LIN {X 0,Y 359.699,Z 331.885,A -85,B 0,C 180,E1 -13391.93,E2 -13391.93} C_VEL
LIN {X 0,Y 358.635,Z 342.585,A -85,B 0,C 180,E1 -13392.906,E2 -13392.906} C_VEL
LIN {X 0,Y 357.527,Z 352.445,A -85,B 0,C 180,E1 -13394.026,E2 -13394.026} C_VEL
LIN {X 0,Y 356.534,Z 362.461,A -85,B 0,C 180,E1 -13395.444,E2 -13395.444} C_VEL
LIN {X 0,Y 355.478,Z 372.178,A -85,B 0,C 180,E1 -13397.149,E2 -13397.149} C_VEL
LIN {X 0,Y 354.559,Z 379.917,A -85,B 0,C 180,E1 -13398.857,E2 -13398.857} C_VEL
LIN {X 0,Y 354.087,Z 385.232,A -85,B 0,C 180,E1 -13400.287,E2 -13400.287} C_VEL
LIN {X 0,Y 353.658,Z 390.386,A -85,B 0,C 180,E1 -13402.004,E2 -13402.004} C_VEL
LIN {X 0,Y 353.447,Z 394.607,A -85,B 0,C 180,E1 -13403.832,E2 -13403.832} C_VEL
LIN {X 0,Y 353.36,Z 397.364,A -85,B 0,C 180,E1 -13405.437,E2 -13405.437} C_VEL
LIN {X 0,Y 353.319,Z 399.786,A -85,B 0,C 180,E1 -13407.72,E2 -13407.72} C_VEL
LIN {X 0,Y 353.4,Z 400.407,A -85,B 0,C 180,E1 -13408.861,E2 -13408.861} C_VEL
LIN {X 0,Y 353.411,Z 400.626,A -85,B 0,C 180,E1 -13410,E2 -13410} C_VEL
LIN {X 0,Y 353.4,Z 400.405,A -85,B 0,C 180,E1 -13411.14,E2 -13411.14} C_VEL
LIN {X 0,Y 353.283,Z 398.772,A -85,B 0,C 180,E1 -13413.422,E2 -13413.422} C_VEL
LIN {X 0,Y 353.36,Z 397.36,A -85,B 0,C 180,E1 -13414.563,E2 -13414.563} C_VEL
LIN {X 0,Y 353.446,Z 394.601,A -85,B 0,C 180,E1 -13416.167,E2 -13416.167} C_VEL
LIN {X 0,Y 353.654,Z 390.371,A -85,B 0,C 180,E1 -13417.996,E2 -13417.996} C_VEL
LIN {X 0,Y 354.203,Z 384.208,A -85,B 0,C 180,E1 -13419.998,E2 -13419.998} C_VEL
LIN {X 0,Y 354.818,Z 377.479,A -85,B 0,C 180,E1 -13421.714,E2 -13421.714} C_VEL
LIN {X 0,Y 355.819,Z 369.151,A -85,B 0,C 180,E1 -13423.42,E2 -13423.42} C_VEL
LIN {X 0,Y 356.807,Z 360.618,A -85,B 0,C 180,E1 -13424.837,E2 -13424.837} C_VEL
LIN {X 0,Y 357.753,Z 350.071,A -85,B 0,C 180,E1 -13426.257,E2 -13426.257} C_VEL
LIN {X 0,Y 359.082,Z 338.231,A -85,B 0,C 180,E1 -13427.513,E2 -13427.513} C_VEL
LIN {X 0,Y 359.668,Z 330.019,A -85,B 0,C 180,E1 -13428.219,E2 -13428.219} C_VEL
LIN {X 0,Y 358.496,Z 318.284,A -85,B 0,C 180,E1 -13429.127,E2 -13429.127} C_VEL
LIN {X 0,Y 356.685,Z 305.211,A -85,B 0,C 180,E1 -13429.919,E2 -13429.919} C_VEL
LIN {X 0,Y 354.401,Z 292.638,A -85,B 0,C 180,E1 -13430.496,E2 -13430.496} C_VEL
LIN {X 0,Y 354.931,Z 285.811,A -85,B 0,C 180,E1 -13433.871,E2 -13433.871} C_VEL
LIN {X 0,Y 355.677,Z 278.035,A -85,B 0,C 180,E1 -13437.688,E2 -13437.688} C_VEL
LIN {X 0,Y 356.457,Z 270.436,A -85,B 0,C 180,E1 -13441.463,E2 -13441.463} C_VEL
LIN {X 0,Y 357.26,Z 263.905,A -85,B 0,C 180,E1 -13444.785,E2 -13444.785} C_VEL
LIN {X 0,Y 357.475,Z 260.008,A -85,B 0,C 180,E1 -13446.859,E2 -13446.859} C_VEL
LIN {X 0,Y 356.766,Z 254.927,A -85,B 0,C 180,E1 -13449.801,E2 -13449.801} C_VEL
LIN {X 0,Y 355.815,Z 249.673,A -85,B 0,C 180,E1 -13453.045,E2 -13453.045} C_VEL
LIN {X 0,Y 354.798,Z 244.294,A -85,B 0,C 180,E1 -13456.67,E2 -13456.67} C_VEL
LIN {X 0,Y 354.787,Z 244.294,A -85,B 0,C 180,E1 -13460.662,E2 -13460.662} C_VEL
LIN {X 0,Y 354.825,Z 244.287,A -85,B 0,C 180,E1 -13464.301,E2 -13464.301} C_VEL
LIN {X 0,Y 354.79,Z 244.288,A -85,B 0,C 180,E1 -13467.667,E2 -13467.667} C_VEL
LIN {X 0,Y 354.802,Z 244.287,A -85,B 0,C 180,E1 -13471.615,E2 -13471.615} C_VEL
LIN {X 0,Y 354.807,Z 244.286,A -85,B 0,C 180,E1 -13475.42,E2 -13475.42} C_VEL
LIN {X 0,Y 354.83,Z 244.283,A -85,B 0,C 180,E1 -13479.113,E2 -13479.113} C_VEL
LIN {X 0,Y 354.903,Z 244.274,A -85,B 0,C 180,E1 -13482.72,E2 -13482.72} C_VEL
LIN {X 0,Y 354.955,Z 244.27,A -85,B 0,C 180,E1 -13486.255,E2 -13486.255} C_VEL
LIN {X 0,Y 354.955,Z 244.273,A -85,B 0,C 180,E1 -13489.735,E2 -13489.735} C_VEL
LIN {X 0,Y 355.116,Z 244.248,A -85,B 0,C 180,E1 -13493.18,E2 -13493.18} C_VEL
LIN {X 0,Y 355.248,Z 244.235,A -85,B 0,C 180,E1 -13497.732,E2 -13497.732} C_VEL
LIN {X 0,Y 355.235,Z 244.232,A -85,B 0,C 180,E1 -13502.268,E2 -13502.268} C_VEL
LIN {X 0,Y 355.116,Z 244.249,A -85,B 0,C 180,E1 -13506.82,E2 -13506.82} C_VEL
LIN {X 0,Y 354.961,Z 244.266,A -85,B 0,C 180,E1 -13510.265,E2 -13510.265} C_VEL
LIN {X 0,Y 354.947,Z 244.268,A -85,B 0,C 180,E1 -13514.019,E2 -13514.019} C_VEL
LIN {X 0,Y 354.894,Z 244.275,A -85,B 0,C 180,E1 -13518.092,E2 -13518.092} C_VEL
LIN {X 0,Y 354.819,Z 244.285,A -85,B 0,C 180,E1 -13522.107,E2 -13522.107} C_VEL
LIN {X 0,Y 354.824,Z 244.283,A -85,B 0,C 180,E1 -13525.833,E2 -13525.833} C_VEL
LIN {X 0,Y 354.799,Z 244.287,A -85,B 0,C 180,E1 -13529.684,E2 -13529.684} C_VEL
LIN {X 0,Y 354.79,Z 244.292,A -85,B 0,C 180,E1 -13532.333,E2 -13532.333} C_VEL
LIN {X 0,Y 354.825,Z 244.284,A -85,B 0,C 180,E1 -13535.699,E2 -13535.699} C_VEL
LIN {X 0,Y 354.827,Z 244.283,A -85,B 0,C 180,E1 -13539.423,E2 -13539.423} C_VEL
LIN {X 0,Y 354.791,Z 244.288,A -85,B 0,C 180,E1 -13542.867,E2 -13542.867} C_VEL
LIN {X 0,Y 354.77,Z 244.296,A -85,B 0,C 180,E1 -13546.104,E2 -13546.104} C_VEL
LIN {X 0,Y 354.787,Z 244.288,A -85,B 0,C 180,E1 -13549.178,E2 -13549.178} C_VEL
LIN {X 0,Y 354.792,Z 244.289,A -85,B 0,C 180,E1 -13552.406,E2 -13552.406} C_VEL
LIN {X 0,Y 354.645,Z 244.306,A -85,B 0,C 180,E1 -13554.921,E2 -13554.921} C_VEL
LIN {X 0,Y 354.359,Z 244.347,A -85,B 0,C 180,E1 -13557.622,E2 -13557.622} C_VEL
LIN {X 0,Y 354.278,Z 245.084,A -85,B 0,C 180,E1 -13558.95,E2 -13558.95} C_VEL
LIN {X 0,Y 354.196,Z 247.346,A -85,B 0,C 180,E1 -13561.561,E2 -13561.561} C_VEL
LIN {X 0,Y 354.111,Z 249.638,A -85,B 0,C 180,E1 -13564.111,E2 -13564.111} C_VEL
LIN {X 0,Y 354.05,Z 251.97,A -85,B 0,C 180,E1 -13566.609,E2 -13566.609} C_VEL
LIN {X 0,Y 354.016,Z 254.952,A -85,B 0,C 180,E1 -13569.596,E2 -13569.596} C_VEL
LIN {X 0,Y 357.921,Z 268.382,A -85,B 0,C 180,E1 -13570.374,E2 -13570.374} C_VEL
LIN {X 0,Y 360.714,Z 280.036,A -85,B 0,C 180,E1 -13571.221,E2 -13571.221} C_VEL
LIN {X 0,Y 361.289,Z 284.038,A -85,B 0,C 180,E1 -13571.541,E2 -13571.541} C_VEL
LIN {X 0,Y 360.357,Z 296.417,A -85,B 0,C 180,E1 -13572.551,E2 -13572.551} C_VEL
LIN {X 0,Y 359.482,Z 306.713,A -85,B 0,C 180,E1 -13573.635,E2 -13573.635} C_VEL
LIN {X 0,Y 358.447,Z 316.732,A -85,B 0,C 180,E1 -13574.942,E2 -13574.942} C_VEL
LIN {X 0,Y 357.377,Z 325.539,A -85,B 0,C 180,E1 -13576.35,E2 -13576.35} C_VEL
LIN {X 0,Y 356.259,Z 334.126,A -85,B 0,C 180,E1 -13578.045,E2 -13578.045} C_VEL
LIN {X 0,Y 355.393,Z 340.963,A -85,B 0,C 180,E1 -13579.748,E2 -13579.748} C_VEL
LIN {X 0,Y 354.749,Z 346.43,A -85,B 0,C 180,E1 -13581.455,E2 -13581.455} C_VEL
LIN {X 0,Y 354.307,Z 350.717,A -85,B 0,C 180,E1 -13583.164,E2 -13583.164} C_VEL
LIN {X 0,Y 353.962,Z 352.992,A -85,B 0,C 180,E1 -13584.302,E2 -13584.302} C_VEL
LIN {X 0,Y 353.832,Z 354.833,A -85,B 0,C 180,E1 -13585.443,E2 -13585.443} C_VEL
LIN {X 0,Y 353.805,Z 356.215,A -85,B 0,C 180,E1 -13586.583,E2 -13586.583} C_VEL
LIN {X 0,Y 353.512,Z 357.818,A -85,B 0,C 180,E1 -13588.861,E2 -13588.861} C_VEL
LIN {X 0,Y 353.483,Z 358.049,A -85,B 0,C 180,E1 -13590,E2 -13590} C_VEL
LIN {X 0,Y 353.634,Z 357.275,A -85,B 0,C 180,E1 -13592.278,E2 -13592.278} C_VEL
LIN {X 0,Y 353.783,Z 356.312,A -85,B 0,C 180,E1 -13593.416,E2 -13593.416} C_VEL
LIN {X 0,Y 353.822,Z 354.972,A -85,B 0,C 180,E1 -13594.557,E2 -13594.557} C_VEL
LIN {X 0,Y 354.111,Z 352.127,A -85,B 0,C 180,E1 -13596.267,E2 -13596.267} C_VEL
LIN {X 0,Y 354.551,Z 348.265,A -85,B 0,C 180,E1 -13597.976,E2 -13597.976} C_VEL
LIN {X 0,Y 355.108,Z 343.282,A -85,B 0,C 180,E1 -13599.685,E2 -13599.685} C_VEL
LIN {X 0,Y 355.96,Z 336.996,A -85,B 0,C 180,E1 -13601.387,E2 -13601.387} C_VEL
LIN {X 0,Y 356.932,Z 329.129,A -85,B 0,C 180,E1 -13603.087,E2 -13603.087} C_VEL
LIN {X 0,Y 357.867,Z 321.104,A -85,B 0,C 180,E1 -13604.501,E2 -13604.501} C_VEL
LIN {X 0,Y 358.993,Z 311.302,A -85,B 0,C 180,E1 -13605.907,E2 -13605.907} C_VEL
LIN {X 0,Y 359.9,Z 301.655,A -85,B 0,C 180,E1 -13607.032,E2 -13607.032} C_VEL
LIN {X 0,Y 360.833,Z 291.2,A -85,B 0,C 180,E1 -13608.011,E2 -13608.011} C_VEL
LIN {X 0,Y 361.263,Z 282.387,A -85,B 0,C 180,E1 -13608.688,E2 -13608.688} C_VEL
LIN {X 0,Y 358.303,Z 269.681,A -85,B 0,C 180,E1 -13609.644,E2 -13609.644} C_VEL
LIN {X 0,Y 354.312,Z 256.261,A -85,B 0,C 180,E1 -13610.444,E2 -13610.444} C_VEL
LIN {X 0,Y 354.04,Z 254.897,A -85,B 0,C 180,E1 -13610.509,E2 -13610.509} C_VEL
LIN {X 0,Y 354.071,Z 250.911,A -85,B 0,C 180,E1 -13614.635,E2 -13614.635} C_VEL
LIN {X 0,Y 354.183,Z 247.453,A -85,B 0,C 180,E1 -13618.439,E2 -13618.439} C_VEL
LIN {X 0,Y 354.294,Z 244.842,A -85,B 0,C 180,E1 -13621.463,E2 -13621.463} C_VEL
LIN {X 0,Y 354.342,Z 244.351,A -85,B 0,C 180,E1 -13622.379,E2 -13622.379} C_VEL
LIN {X 0,Y 354.712,Z 244.299,A -85,B 0,C 180,E1 -13625.674,E2 -13625.674} C_VEL
LIN {X 0,Y 354.763,Z 244.292,A -85,B 0,C 180,E1 -13627.302,E2 -13627.302} C_VEL
LIN {X 0,Y 354.156,Z 244.373,A -85,B 0,C 180,E1 -13628.25,E2 -13628.25} C_VEL
LIN {X 0,Y 351.326,Z 244.724,A -85,B 0,C 180,E1 -13629.791,E2 -13629.791} C_VEL
LIN {X 0,Y 348.881,Z 245.028,A -85,B 0,C 180,E1 -13631.038,E2 -13631.038} C_VEL
LIN {X 0,Y 347.812,Z 245.162,A -85,B 0,C 180,E1 -13632.003,E2 -13632.003} C_VEL
LIN {X 0,Y 347.717,Z 245.168,A -85,B 0,C 180,E1 -13632.33,E2 -13632.33} C_VEL
LIN {X 0,Y 347.707,Z 245.17,A -85,B 0,C 180,E1 -13635.027,E2 -13635.027} C_VEL
LIN {X 0,Y 347.751,Z 245.166,A -85,B 0,C 180,E1 -13638.397,E2 -13638.397} C_VEL
LIN {X 0,Y 347.774,Z 245.165,A -85,B 0,C 180,E1 -13642.011,E2 -13642.011} C_VEL
LIN {X 0,Y 347.746,Z 245.17,A -85,B 0,C 180,E1 -13645.536,E2 -13645.536} C_VEL
LIN {X 0,Y 347.748,Z 245.165,A -85,B 0,C 180,E1 -13648.301,E2 -13648.301} C_VEL
LIN {X 0,Y 347.747,Z 245.166,A -85,B 0,C 180,E1 -13650.985,E2 -13650.985} C_VEL
LIN {X 0,Y 347.752,Z 245.168,A -85,B 0,C 180,E1 -13653.601,E2 -13653.601} C_VEL
LIN {X 0,Y 347.772,Z 245.162,A -85,B 0,C 180,E1 -13656.161,E2 -13656.161} C_VEL
LIN {X 0,Y 347.802,Z 245.159,A -85,B 0,C 180,E1 -13659.909,E2 -13659.909} C_VEL
LIN {X 0,Y 347.833,Z 245.156,A -85,B 0,C 180,E1 -13663.568,E2 -13663.568} C_VEL
LIN {X 0,Y 347.893,Z 245.151,A -85,B 0,C 180,E1 -13667.161,E2 -13667.161} C_VEL
LIN {X 0,Y 348.096,Z 245.122,A -85,B 0,C 180,E1 -13671.612,E2 -13671.612} C_VEL
LIN {X 0,Y 348.067,Z 245.126,A -85,B 0,C 180,E1 -13674.206,E2 -13674.206} C_VEL
LIN {X 0,Y 348.196,Z 245.109,A -85,B 0,C 180,E1 -13677.686,E2 -13677.686} C_VEL
LIN {X 0,Y 348.147,Z 245.116,A -85,B 0,C 180,E1 -13681.157,E2 -13681.157} C_VEL
LIN {X 0,Y 348.208,Z 245.112,A -85,B 0,C 180,E1 -13682.313,E2 -13682.313} C_VEL
LIN {X 0,Y 348.08,Z 245.124,A -85,B 0,C 180,E1 -13686.958,E2 -13686.958} C_VEL
LIN {X 0,Y 347.895,Z 245.15,A -85,B 0,C 180,E1 -13690.475,E2 -13690.475} C_VEL
LIN {X 0,Y 347.901,Z 245.152,A -85,B 0,C 180,E1 -13694.15,E2 -13694.15} C_VEL
LIN {X 0,Y 347.894,Z 245.15,A -85,B 0,C 180,E1 -13698.291,E2 -13698.291} C_VEL
LIN {X 0,Y 347.766,Z 245.166,A -85,B 0,C 180,E1 -13701.625,E2 -13701.625} C_VEL
LIN {X 0,Y 347.739,Z 245.167,A -85,B 0,C 180,E1 -13705.114,E2 -13705.114} C_VEL
LIN {X 0,Y 347.737,Z 245.173,A -85,B 0,C 180,E1 -13707.7,E2 -13707.7} C_VEL
LIN {X 0,Y 347.742,Z 245.167,A -85,B 0,C 180,E1 -13710.349,E2 -13710.349} C_VEL
LIN {X 0,Y 347.75,Z 245.167,A -85,B 0,C 180,E1 -13714.044,E2 -13714.044} C_VEL
LIN {X 0,Y 347.757,Z 245.17,A -85,B 0,C 180,E1 -13717.321,E2 -13717.321} C_VEL
LIN {X 0,Y 347.742,Z 245.169,A -85,B 0,C 180,E1 -13721.601,E2 -13721.601} C_VEL
LIN {X 0,Y 347.769,Z 245.276,A -85,B 0,C 180,E1 -13722.971,E2 -13722.971} C_VEL
LIN {X 0,Y 348.742,Z 250.485,A -85,B 0,C 180,E1 -13726.51,E2 -13726.51} C_VEL
LIN {X 0,Y 349.745,Z 256,A -85,B 0,C 180,E1 -13729.982,E2 -13729.982} C_VEL
LIN {X 0,Y 350.464,Z 261.145,A -85,B 0,C 180,E1 -13733.015,E2 -13733.015} C_VEL
LIN {X 0,Y 350.204,Z 265.441,A -85,B 0,C 180,E1 -13735.366,E2 -13735.366} C_VEL
LIN {X 0,Y 349.297,Z 272.644,A -85,B 0,C 180,E1 -13739.131,E2 -13739.131} C_VEL
LIN {X 0,Y 348.563,Z 279.286,A -85,B 0,C 180,E1 -13742.519,E2 -13742.519} C_VEL
LIN {X 0,Y 347.839,Z 286.516,A -85,B 0,C 180,E1 -13746.166,E2 -13746.166} C_VEL
LIN {X 0,Y 347.376,Z 292.278,A -85,B 0,C 180,E1 -13749.071,E2 -13749.071} C_VEL
LIN {X 0,Y 349.887,Z 305.889,A -85,B 0,C 180,E1 -13749.717,E2 -13749.717} C_VEL
LIN {X 0,Y 351.591,Z 318.635,A -85,B 0,C 180,E1 -13750.527,E2 -13750.527} C_VEL
LIN {X 0,Y 352.663,Z 329.662,A -85,B 0,C 180,E1 -13751.406,E2 -13751.406} C_VEL
LIN {X 0,Y 352.791,Z 333.152,A -85,B 0,C 180,E1 -13751.714,E2 -13751.714} C_VEL
LIN {X 0,Y 351.522,Z 344.774,A -85,B 0,C 180,E1 -13752.849,E2 -13752.849} C_VEL
LIN {X 0,Y 350.29,Z 355.459,A -85,B 0,C 180,E1 -13754.165,E2 -13754.165} C_VEL
LIN {X 0,Y 349.416,Z 363.829,A -85,B 0,C 180,E1 -13755.439,E2 -13755.439} C_VEL
LIN {X 0,Y 348.53,Z 371.751,A -85,B 0,C 180,E1 -13756.888,E2 -13756.888} C_VEL
LIN {X 0,Y 347.551,Z 379.488,A -85,B 0,C 180,E1 -13758.629,E2 -13758.629} C_VEL
LIN {X 0,Y 347.071,Z 384.804,A -85,B 0,C 180,E1 -13760.089,E2 -13760.089} C_VEL
LIN {X 0,Y 346.594,Z 389.958,A -85,B 0,C 180,E1 -13761.84,E2 -13761.84} C_VEL
LIN {X 0,Y 346.343,Z 394.513,A -85,B 0,C 180,E1 -13763.886,E2 -13763.886} C_VEL
LIN {X 0,Y 346.274,Z 396.936,A -85,B 0,C 180,E1 -13765.344,E2 -13765.344} C_VEL
LIN {X 0,Y 346.224,Z 399.358,A -85,B 0,C 180,E1 -13767.673,E2 -13767.673} C_VEL
LIN {X 0,Y 346.32,Z 399.98,A -85,B 0,C 180,E1 -13768.837,E2 -13768.837} C_VEL
LIN {X 0,Y 346.35,Z 400.2,A -85,B 0,C 180,E1 -13770,E2 -13770} C_VEL
LIN {X 0,Y 346.32,Z 399.978,A -85,B 0,C 180,E1 -13771.163,E2 -13771.163} C_VEL
LIN {X 0,Y 346.206,Z 398.345,A -85,B 0,C 180,E1 -13773.492,E2 -13773.492} C_VEL
LIN {X 0,Y 346.274,Z 396.932,A -85,B 0,C 180,E1 -13774.657,E2 -13774.657} C_VEL
LIN {X 0,Y 346.343,Z 394.506,A -85,B 0,C 180,E1 -13776.113,E2 -13776.113} C_VEL
LIN {X 0,Y 346.592,Z 389.94,A -85,B 0,C 180,E1 -13778.16,E2 -13778.16} C_VEL
LIN {X 0,Y 347.172,Z 383.777,A -85,B 0,C 180,E1 -13780.203,E2 -13780.203} C_VEL
LIN {X 0,Y 347.831,Z 377.048,A -85,B 0,C 180,E1 -13781.953,E2 -13781.953} C_VEL
LIN {X 0,Y 348.846,Z 368.717,A -85,B 0,C 180,E1 -13783.693,E2 -13783.693} C_VEL
LIN {X 0,Y 350.015,Z 359.161,A -85,B 0,C 180,E1 -13785.288,E2 -13785.288} C_VEL
LIN {X 0,Y 350.909,Z 349.638,A -85,B 0,C 180,E1 -13786.583,E2 -13786.583} C_VEL
LIN {X 0,Y 352.317,Z 337.799,A -85,B 0,C 180,E1 -13787.861,E2 -13787.861} C_VEL
LIN {X 0,Y 352.813,Z 331.363,A -85,B 0,C 180,E1 -13788.435,E2 -13788.435} C_VEL
LIN {X 0,Y 351.787,Z 320.21,A -85,B 0,C 180,E1 -13789.349,E2 -13789.349} C_VEL
LIN {X 0,Y 350.003,Z 306.683,A -85,B 0,C 180,E1 -13790.228,E2 -13790.228} C_VEL
LIN {X 0,Y 347.564,Z 293.686,A -85,B 0,C 180,E1 -13790.869,E2 -13790.869} C_VEL
LIN {X 0,Y 347.392,Z 292.22,A -85,B 0,C 180,E1 -13790.919,E2 -13790.919} C_VEL
LIN {X 0,Y 348.091,Z 283.999,A -85,B 0,C 180,E1 -13795.087,E2 -13795.087} C_VEL
LIN {X 0,Y 348.873,Z 276.433,A -85,B 0,C 180,E1 -13798.913,E2 -13798.913} C_VEL
LIN {X 0,Y 349.772,Z 268.732,A -85,B 0,C 180,E1 -13802.855,E2 -13802.855} C_VEL
LIN {X 0,Y 350.378,Z 263.584,A -85,B 0,C 180,E1 -13805.57,E2 -13805.57} C_VEL
LIN {X 0,Y 350.337,Z 259.724,A -85,B 0,C 180,E1 -13807.724,E2 -13807.724} C_VEL
LIN {X 0,Y 349.539,Z 254.573,A -85,B 0,C 180,E1 -13810.835,E2 -13810.835} C_VEL
LIN {X 0,Y 348.371,Z 248.298,A -85,B 0,C 180,E1 -13814.918,E2 -13814.918} C_VEL
LIN {X 0,Y 347.755,Z 245.17,A -85,B 0,C 180,E1 -13817.219,E2 -13817.219} C_VEL
LIN {X 0,Y 347.733,Z 245.168,A -85,B 0,C 180,E1 -13821.205,E2 -13821.205} C_VEL
LIN {X 0,Y 347.791,Z 245.162,A -85,B 0,C 180,E1 -13824.125,E2 -13824.125} C_VEL
LIN {X 0,Y 347.742,Z 245.169,A -85,B 0,C 180,E1 -13828.086,E2 -13828.086} C_VEL
LIN {X 0,Y 347.748,Z 245.166,A -85,B 0,C 180,E1 -13830.985,E2 -13830.985} C_VEL
LIN {X 0,Y 347.745,Z 245.166,A -85,B 0,C 180,E1 -13833.601,E2 -13833.601} C_VEL
LIN {X 0,Y 347.752,Z 245.171,A -85,B 0,C 180,E1 -13836.159,E2 -13836.159} C_VEL
LIN {X 0,Y 347.812,Z 245.162,A -85,B 0,C 180,E1 -13839.909,E2 -13839.909} C_VEL
LIN {X 0,Y 347.87,Z 245.153,A -85,B 0,C 180,E1 -13842.359,E2 -13842.359} C_VEL
LIN {X 0,Y 347.901,Z 245.151,A -85,B 0,C 180,E1 -13845.971,E2 -13845.971} C_VEL
LIN {X 0,Y 347.895,Z 245.15,A -85,B 0,C 180,E1 -13849.525,E2 -13849.525} C_VEL
LIN {X 0,Y 348.082,Z 245.124,A -85,B 0,C 180,E1 -13853.042,E2 -13853.042} C_VEL
LIN {X 0,Y 348.21,Z 245.112,A -85,B 0,C 180,E1 -13857.687,E2 -13857.687} C_VEL
LIN {X 0,Y 348.121,Z 245.121,A -85,B 0,C 180,E1 -13861.157,E2 -13861.157} C_VEL
LIN {X 0,Y 348.197,Z 245.109,A -85,B 0,C 180,E1 -13862.314,E2 -13862.314} C_VEL
LIN {X 0,Y 348.082,Z 245.126,A -85,B 0,C 180,E1 -13866.958,E2 -13866.958} C_VEL
LIN {X 0,Y 347.901,Z 245.146,A -85,B 0,C 180,E1 -13870.475,E2 -13870.475} C_VEL
LIN {X 0,Y 347.903,Z 245.146,A -85,B 0,C 180,E1 -13874.15,E2 -13874.15} C_VEL
LIN {X 0,Y 347.833,Z 245.155,A -85,B 0,C 180,E1 -13878.259,E2 -13878.259} C_VEL
LIN {X 0,Y 347.771,Z 245.162,A -85,B 0,C 180,E1 -13881.626,E2 -13881.626} C_VEL
LIN {X 0,Y 347.776,Z 245.163,A -85,B 0,C 180,E1 -13885.111,E2 -13885.111} C_VEL
LIN {X 0,Y 347.741,Z 245.166,A -85,B 0,C 180,E1 -13887.7,E2 -13887.7} C_VEL
LIN {X 0,Y 347.741,Z 245.17,A -85,B 0,C 180,E1 -13890.349,E2 -13890.349} C_VEL
LIN {X 0,Y 347.752,Z 245.167,A -85,B 0,C 180,E1 -13894.044,E2 -13894.044} C_VEL
LIN {X 0,Y 347.764,Z 245.163,A -85,B 0,C 180,E1 -13897.321,E2 -13897.321} C_VEL
LIN {X 0,Y 347.735,Z 245.172,A -85,B 0,C 180,E1 -13900.297,E2 -13900.297} C_VEL
LIN {X 0,Y 347.726,Z 245.168,A -85,B 0,C 180,E1 -13903.408,E2 -13903.408} C_VEL
LIN {X 0,Y 347.728,Z 245.168,A -85,B 0,C 180,E1 -13906.686,E2 -13906.686} C_VEL
LIN {X 0,Y 347.749,Z 245.168,A -85,B 0,C 180,E1 -13910.173,E2 -13910.173} C_VEL
LIN {X 0,Y 347.739,Z 245.166,A -85,B 0,C 180,E1 -13912.676,E2 -13912.676} C_VEL
LIN {X 0,Y 347.486,Z 245.202,A -85,B 0,C 180,E1 -13916.021,E2 -13916.021} C_VEL
LIN {X 0,Y 347.269,Z 245.446,A -85,B 0,C 180,E1 -13918.252,E2 -13918.252} C_VEL
LIN {X 0,Y 347.192,Z 247.715,A -85,B 0,C 180,E1 -13920.934,E2 -13920.934} C_VEL
LIN {X 0,Y 347.103,Z 250.029,A -85,B 0,C 180,E1 -13923.548,E2 -13923.548} C_VEL
LIN {X 0,Y 347.045,Z 252.379,A -85,B 0,C 180,E1 -13926.107,E2 -13926.107} C_VEL
LIN {X 0,Y 347.001,Z 255.445,A -85,B 0,C 180,E1 -13929.169,E2 -13929.169} C_VEL
LIN {X 0,Y 350.855,Z 268.565,A -85,B 0,C 180,E1 -13929.948,E2 -13929.948} C_VEL
LIN {X 0,Y 353.896,Z 280.989,A -85,B 0,C 180,E1 -13930.879,E2 -13930.879} C_VEL
LIN {X 0,Y 354.572,Z 284.714,A -85,B 0,C 180,E1 -13931.197,E2 -13931.197} C_VEL
LIN {X 0,Y 353.624,Z 296.848,A -85,B 0,C 180,E1 -13932.207,E2 -13932.207} C_VEL
LIN {X 0,Y 352.659,Z 307.491,A -85,B 0,C 180,E1 -13933.354,E2 -13933.354} C_VEL
LIN {X 0,Y 351.608,Z 317.162,A -85,B 0,C 180,E1 -13934.642,E2 -13934.642} C_VEL
LIN {X 0,Y 350.477,Z 325.969,A -85,B 0,C 180,E1 -13936.076,E2 -13936.076} C_VEL
LIN {X 0,Y 349.336,Z 334.554,A -85,B 0,C 180,E1 -13937.805,E2 -13937.805} C_VEL
LIN {X 0,Y 348.421,Z 341.391,A -85,B 0,C 180,E1 -13939.54,E2 -13939.54} C_VEL
LIN {X 0,Y 347.756,Z 346.858,A -85,B 0,C 180,E1 -13941.282,E2 -13941.282} C_VEL
LIN {X 0,Y 347.282,Z 351.145,A -85,B 0,C 180,E1 -13943.026,E2 -13943.026} C_VEL
LIN {X 0,Y 346.926,Z 353.419,A -85,B 0,C 180,E1 -13944.186,E2 -13944.186} C_VEL
LIN {X 0,Y 346.759,Z 355.261,A -85,B 0,C 180,E1 -13945.35,E2 -13945.35} C_VEL
LIN {X 0,Y 346.735,Z 356.642,A -85,B 0,C 180,E1 -13946.514,E2 -13946.514} C_VEL
LIN {X 0,Y 346.45,Z 358.243,A -85,B 0,C 180,E1 -13948.837,E2 -13948.837} C_VEL
LIN {X 0,Y 346.419,Z 358.475,A -85,B 0,C 180,E1 -13950,E2 -13950} C_VEL
LIN {X 0,Y 346.579,Z 357.7,A -85,B 0,C 180,E1 -13952.324,E2 -13952.324} C_VEL
LIN {X 0,Y 346.714,Z 356.738,A -85,B 0,C 180,E1 -13953.486,E2 -13953.486} C_VEL
LIN {X 0,Y 346.748,Z 355.399,A -85,B 0,C 180,E1 -13954.65,E2 -13954.65} C_VEL
LIN {X 0,Y 347.083,Z 352.551,A -85,B 0,C 180,E1 -13956.394,E2 -13956.394} C_VEL
LIN {X 0,Y 347.524,Z 348.691,A -85,B 0,C 180,E1 -13958.138,E2 -13958.138} C_VEL
LIN {X 0,Y 348.111,Z 343.708,A -85,B 0,C 180,E1 -13959.881,E2 -13959.881} C_VEL
LIN {X 0,Y 349.017,Z 337.421,A -85,B 0,C 180,E1 -13961.617,E2 -13961.617} C_VEL
LIN {X 0,Y 350.044,Z 329.552,A -85,B 0,C 180,E1 -13963.349,E2 -13963.349} C_VEL
LIN {X 0,Y 351.019,Z 321.527,A -85,B 0,C 180,E1 -13964.79,E2 -13964.79} C_VEL
LIN {X 0,Y 352.19,Z 311.724,A -85,B 0,C 180,E1 -13966.223,E2 -13966.223} C_VEL
LIN {X 0,Y 353.129,Z 302.077,A -85,B 0,C 180,E1 -13967.369,E2 -13967.369} C_VEL
LIN {X 0,Y 354.113,Z 291.619,A -85,B 0,C 180,E1 -13968.365,E2 -13968.365} C_VEL
LIN {X 0,Y 354.608,Z 284.317,A -85,B 0,C 180,E1 -13968.936,E2 -13968.936} C_VEL
LIN {X 0,Y 351.729,Z 271.686,A -85,B 0,C 180,E1 -13969.944,E2 -13969.944} C_VEL
LIN {X 0,Y 348.006,Z 258.847,A -85,B 0,C 180,E1 -13970.757,E2 -13970.757} C_VEL
LIN {X 0,Y 346.974,Z 255.305,A -85,B 0,C 180,E1 -13970.967,E2 -13970.967} C_VEL
LIN {X 0,Y 347.039,Z 252.095,A -85,B 0,C 180,E1 -13974.312,E2 -13974.312} C_VEL
LIN {X 0,Y 347.104,Z 248.978,A -85,B 0,C 180,E1 -13977.755,E2 -13977.755} C_VEL
LIN {X 0,Y 347.197,Z 246.68,A -85,B 0,C 180,E1 -13980.401,E2 -13980.401} C_VEL
LIN {X 0,Y 347.252,Z 245.516,A -85,B 0,C 180,E1 -13981.784,E2 -13981.784} C_VEL
LIN {X 0,Y 347.549,Z 245.195,A -85,B 0,C 180,E1 -13984.486,E2 -13984.486} C_VEL
LIN {X 0,Y 347.738,Z 245.167,A -85,B 0,C 180,E1 -13987.324,E2 -13987.324} C_VEL
LIN {X 0,Y 347.734,Z 245.171,A -85,B 0,C 180,E1 -13990.297,E2 -13990.297} C_VEL
LIN {X 0,Y 347.717,Z 245.168,A -85,B 0,C 180,E1 -13992.33,E2 -13992.33} C_VEL
LIN {X 0,Y 347.027,Z 245.256,A -85,B 0,C 180,E1 -13993.297,E2 -13993.297} C_VEL
LIN {X 0,Y 344.165,Z 245.612,A -85,B 0,C 180,E1 -13994.87,E2 -13994.87} C_VEL
LIN {X 0,Y 341.766,Z 245.914,A -85,B 0,C 180,E1 -13996.143,E2 -13996.143} C_VEL
LIN {X 0,Y 340.752,Z 246.036,A -85,B 0,C 180,E1 -13997.128,E2 -13997.128} C_VEL
LIN {X 0,Y 340.678,Z 246.047,A -85,B 0,C 180,E1 -13997.462,E2 -13997.462} C_VEL
LIN {X 0,Y 340.701,Z 246.045,A -85,B 0,C 180,E1 -14000.247,E2 -14000.247} C_VEL
LIN {X 0,Y 340.712,Z 246.046,A -85,B 0,C 180,E1 -14003.559,E2 -14003.559} C_VEL
LIN {X 0,Y 340.696,Z 246.045,A -85,B 0,C 180,E1 -14006.154,E2 -14006.154} C_VEL
LIN {X 0,Y 340.725,Z 246.041,A -85,B 0,C 180,E1 -14010.034,E2 -14010.034} C_VEL
LIN {X 0,Y 340.722,Z 246.042,A -85,B 0,C 180,E1 -14013.013,E2 -14013.013} C_VEL
LIN {X 0,Y 340.743,Z 246.041,A -85,B 0,C 180,E1 -14015.637,E2 -14015.637} C_VEL
LIN {X 0,Y 340.732,Z 246.042,A -85,B 0,C 180,E1 -14019.473,E2 -14019.473} C_VEL
LIN {X 0,Y 340.794,Z 246.031,A -85,B 0,C 180,E1 -14021.981,E2 -14021.981} C_VEL
LIN {X 0,Y 340.871,Z 246.022,A -85,B 0,C 180,E1 -14025.705,E2 -14025.705} C_VEL
LIN {X 0,Y 340.874,Z 246.023,A -85,B 0,C 180,E1 -14029.306,E2 -14029.306} C_VEL
LIN {X 0,Y 341.077,Z 246.001,A -85,B 0,C 180,E1 -14032.898,E2 -14032.898} C_VEL
LIN {X 0,Y 341.133,Z 245.989,A -85,B 0,C 180,E1 -14037.638,E2 -14037.638} C_VEL
LIN {X 0,Y 341.116,Z 245.992,A -85,B 0,C 180,E1 -14041.18,E2 -14041.18} C_VEL
LIN {X 0,Y 341.17,Z 245.989,A -85,B 0,C 180,E1 -14042.361,E2 -14042.361} C_VEL
LIN {X 0,Y 341.048,Z 246,A -85,B 0,C 180,E1 -14047.102,E2 -14047.102} C_VEL
LIN {X 0,Y 340.847,Z 246.027,A -85,B 0,C 180,E1 -14050.695,E2 -14050.695} C_VEL
LIN {X 0,Y 340.865,Z 246.026,A -85,B 0,C 180,E1 -14054.325,E2 -14054.325} C_VEL
LIN {X 0,Y 340.84,Z 246.027,A -85,B 0,C 180,E1 -14058.467,E2 -14058.467} C_VEL
LIN {X 0,Y 340.719,Z 246.046,A -85,B 0,C 180,E1 -14061.842,E2 -14061.842} C_VEL
LIN {X 0,Y 340.676,Z 246.052,A -85,B 0,C 180,E1 -14065.672,E2 -14065.672} C_VEL
LIN {X 0,Y 340.683,Z 246.047,A -85,B 0,C 180,E1 -14068.325,E2 -14068.325} C_VEL
LIN {X 0,Y 340.696,Z 246.046,A -85,B 0,C 180,E1 -14071.045,E2 -14071.045} C_VEL
LIN {X 0,Y 340.719,Z 246.046,A -85,B 0,C 180,E1 -14075.279,E2 -14075.279} C_VEL
LIN {X 0,Y 340.695,Z 246.045,A -85,B 0,C 180,E1 -14078.382,E2 -14078.382} C_VEL
LIN {X 0,Y 340.731,Z 246.075,A -85,B 0,C 180,E1 -14082.418,E2 -14082.418} C_VEL
LIN {X 0,Y 341.688,Z 251.245,A -85,B 0,C 180,E1 -14086.046,E2 -14086.046} C_VEL
LIN {X 0,Y 342.631,Z 256.348,A -85,B 0,C 180,E1 -14089.371,E2 -14089.371} C_VEL
LIN {X 0,Y 343.328,Z 260.832,A -85,B 0,C 180,E1 -14092.113,E2 -14092.113} C_VEL
LIN {X 0,Y 343.385,Z 264.665,A -85,B 0,C 180,E1 -14094.317,E2 -14094.317} C_VEL
LIN {X 0,Y 342.556,Z 271.031,A -85,B 0,C 180,E1 -14097.763,E2 -14097.763} C_VEL
LIN {X 0,Y 341.678,Z 278.627,A -85,B 0,C 180,E1 -14101.765,E2 -14101.765} C_VEL
LIN {X 0,Y 340.864,Z 286.115,A -85,B 0,C 180,E1 -14105.647,E2 -14105.647} C_VEL
LIN {X 0,Y 340.39,Z 291.854,A -85,B 0,C 180,E1 -14108.62,E2 -14108.62} C_VEL
LIN {X 0,Y 342.92,Z 305.591,A -85,B 0,C 180,E1 -14109.294,E2 -14109.294} C_VEL
LIN {X 0,Y 344.647,Z 318.238,A -85,B 0,C 180,E1 -14110.121,E2 -14110.121} C_VEL
LIN {X 0,Y 345.847,Z 331.016,A -85,B 0,C 180,E1 -14111.18,E2 -14111.18} C_VEL
LIN {X 0,Y 345.707,Z 335.904,A -85,B 0,C 180,E1 -14111.633,E2 -14111.633} C_VEL
LIN {X 0,Y 344.426,Z 346.912,A -85,B 0,C 180,E1 -14112.79,E2 -14112.79} C_VEL
LIN {X 0,Y 343.268,Z 356.263,A -85,B 0,C 180,E1 -14114.016,E2 -14114.016} C_VEL
LIN {X 0,Y 342.291,Z 365.088,A -85,B 0,C 180,E1 -14115.433,E2 -14115.433} C_VEL
LIN {X 0,Y 341.208,Z 374.076,A -85,B 0,C 180,E1 -14117.207,E2 -14117.207} C_VEL
LIN {X 0,Y 340.345,Z 381.316,A -85,B 0,C 180,E1 -14118.988,E2 -14118.988} C_VEL
LIN {X 0,Y 339.846,Z 386.212,A -85,B 0,C 180,E1 -14120.477,E2 -14120.477} C_VEL
LIN {X 0,Y 339.445,Z 390.977,A -85,B 0,C 180,E1 -14122.266,E2 -14122.266} C_VEL
LIN {X 0,Y 339.258,Z 394.625,A -85,B 0,C 180,E1 -14124.055,E2 -14124.055} C_VEL
LIN {X 0,Y 339.194,Z 396.509,A -85,B 0,C 180,E1 -14125.246,E2 -14125.246} C_VEL
LIN {X 0,Y 339.13,Z 397.921,A -85,B 0,C 180,E1 -14126.436,E2 -14126.436} C_VEL
LIN {X 0,Y 339.227,Z 399.553,A -85,B 0,C 180,E1 -14128.813,E2 -14128.813} C_VEL
LIN {X 0,Y 339.29,Z 399.775,A -85,B 0,C 180,E1 -14130,E2 -14130} C_VEL
LIN {X 0,Y 339.227,Z 399.551,A -85,B 0,C 180,E1 -14131.187,E2 -14131.187} C_VEL
LIN {X 0,Y 339.13,Z 397.917,A -85,B 0,C 180,E1 -14133.565,E2 -14133.565} C_VEL
LIN {X 0,Y 339.193,Z 396.503,A -85,B 0,C 180,E1 -14134.754,E2 -14134.754} C_VEL
LIN {X 0,Y 339.298,Z 393.53,A -85,B 0,C 180,E1 -14136.541,E2 -14136.541} C_VEL
LIN {X 0,Y 339.547,Z 389.511,A -85,B 0,C 180,E1 -14138.331,E2 -14138.331} C_VEL
LIN {X 0,Y 340.144,Z 383.345,A -85,B 0,C 180,E1 -14140.416,E2 -14140.416} C_VEL
LIN {X 0,Y 340.862,Z 376.617,A -85,B 0,C 180,E1 -14142.201,E2 -14142.201} C_VEL
LIN {X 0,Y 341.88,Z 368.283,A -85,B 0,C 180,E1 -14143.978,E2 -14143.978} C_VEL
LIN {X 0,Y 343.017,Z 359.753,A -85,B 0,C 180,E1 -14145.448,E2 -14145.448} C_VEL
LIN {X 0,Y 343.937,Z 350.385,A -85,B 0,C 180,E1 -14146.776,E2 -14146.776} C_VEL
LIN {X 0,Y 345.36,Z 338.798,A -85,B 0,C 180,E1 -14148.08,E2 -14148.08} C_VEL
LIN {X 0,Y 345.966,Z 332.635,A -85,B 0,C 180,E1 -14148.66,E2 -14148.66} C_VEL
LIN {X 0,Y 344.937,Z 320.711,A -85,B 0,C 180,E1 -14149.685,E2 -14149.685} C_VEL
LIN {X 0,Y 343.202,Z 307.384,A -85,B 0,C 180,E1 -14150.588,E2 -14150.588} C_VEL
LIN {X 0,Y 340.796,Z 294.148,A -85,B 0,C 180,E1 -14151.276,E2 -14151.276} C_VEL
LIN {X 0,Y 340.374,Z 291.778,A -85,B 0,C 180,E1 -14151.381,E2 -14151.381} C_VEL
LIN {X 0,Y 341.129,Z 283.606,A -85,B 0,C 180,E1 -14155.636,E2 -14155.636} C_VEL
LIN {X 0,Y 341.928,Z 276.069,A -85,B 0,C 180,E1 -14159.558,E2 -14159.558} C_VEL
LIN {X 0,Y 342.712,Z 269.958,A -85,B 0,C 180,E1 -14162.776,E2 -14162.776} C_VEL
LIN {X 0,Y 343.383,Z 264.563,A -85,B 0,C 180,E1 -14165.683,E2 -14165.683} C_VEL
LIN {X 0,Y 343.315,Z 260.722,A -85,B 0,C 180,E1 -14167.889,E2 -14167.889} C_VEL
LIN {X 0,Y 342.51,Z 255.581,A -85,B 0,C 180,E1 -14171.042,E2 -14171.042} C_VEL
LIN {X 0,Y 341.572,Z 250.54,A -85,B 0,C 180,E1 -14174.393,E2 -14174.393} C_VEL
LIN {X 0,Y 340.711,Z 246.049,A -85,B 0,C 180,E1 -14177.698,E2 -14177.698} C_VEL
LIN {X 0,Y 340.721,Z 246.04,A -85,B 0,C 180,E1 -14181.771,E2 -14181.771} C_VEL
LIN {X 0,Y 340.726,Z 246.04,A -85,B 0,C 180,E1 -14185.596,E2 -14185.596} C_VEL
LIN {X 0,Y 340.697,Z 246.045,A -85,B 0,C 180,E1 -14188.955,E2 -14188.955} C_VEL
LIN {X 0,Y 340.72,Z 246.041,A -85,B 0,C 180,E1 -14193.013,E2 -14193.013} C_VEL
LIN {X 0,Y 340.704,Z 246.044,A -85,B 0,C 180,E1 -14196.925,E2 -14196.925} C_VEL
LIN {X 0,Y 340.794,Z 246.032,A -85,B 0,C 180,E1 -14200.734,E2 -14200.734} C_VEL
LIN {X 0,Y 340.79,Z 246.032,A -85,B 0,C 180,E1 -14203.219,E2 -14203.219} C_VEL
LIN {X 0,Y 340.846,Z 246.025,A -85,B 0,C 180,E1 -14206.891,E2 -14206.891} C_VEL
LIN {X 0,Y 340.884,Z 246.02,A -85,B 0,C 180,E1 -14210.507,E2 -14210.507} C_VEL
LIN {X 0,Y 341.05,Z 245.999,A -85,B 0,C 180,E1 -14212.898,E2 -14212.898} C_VEL
LIN {X 0,Y 341.172,Z 245.989,A -85,B 0,C 180,E1 -14217.639,E2 -14217.639} C_VEL
LIN {X 0,Y 341.092,Z 245.997,A -85,B 0,C 180,E1 -14221.181,E2 -14221.181} C_VEL
LIN {X 0,Y 341.134,Z 245.989,A -85,B 0,C 180,E1 -14222.362,E2 -14222.362} C_VEL
LIN {X 0,Y 341.049,Z 246.003,A -85,B 0,C 180,E1 -14227.102,E2 -14227.102} C_VEL
LIN {X 0,Y 340.853,Z 246.026,A -85,B 0,C 180,E1 -14230.694,E2 -14230.694} C_VEL
LIN {X 0,Y 340.867,Z 246.023,A -85,B 0,C 180,E1 -14234.325,E2 -14234.325} C_VEL
LIN {X 0,Y 340.789,Z 246.033,A -85,B 0,C 180,E1 -14238.44,E2 -14238.44} C_VEL
LIN {X 0,Y 340.721,Z 246.04,A -85,B 0,C 180,E1 -14241.842,E2 -14241.842} C_VEL
LIN {X 0,Y 340.727,Z 246.039,A -85,B 0,C 180,E1 -14245.668,E2 -14245.668} C_VEL
LIN {X 0,Y 340.708,Z 246.042,A -85,B 0,C 180,E1 -14249.674,E2 -14249.674} C_VEL
LIN {X 0,Y 340.689,Z 246.05,A -85,B 0,C 180,E1 -14252.436,E2 -14252.436} C_VEL
LIN {X 0,Y 340.721,Z 246.04,A -85,B 0,C 180,E1 -14255.279,E2 -14255.279} C_VEL
LIN {X 0,Y 340.713,Z 246.046,A -85,B 0,C 180,E1 -14258.386,E2 -14258.386} C_VEL
LIN {X 0,Y 340.702,Z 246.048,A -85,B 0,C 180,E1 -14262.045,E2 -14262.045} C_VEL
LIN {X 0,Y 340.655,Z 246.052,A -85,B 0,C 180,E1 -14266.227,E2 -14266.227} C_VEL
LIN {X 0,Y 340.689,Z 246.049,A -85,B 0,C 180,E1 -14269.753,E2 -14269.753} C_VEL
LIN {X 0,Y 340.727,Z 246.044,A -85,B 0,C 180,E1 -14271.771,E2 -14271.771} C_VEL
LIN {X 0,Y 340.554,Z 246.061,A -85,B 0,C 180,E1 -14274.701,E2 -14274.701} C_VEL
LIN {X 0,Y 340.216,Z 246.109,A -85,B 0,C 180,E1 -14277.883,E2 -14277.883} C_VEL
LIN {X 0,Y 340.107,Z 249.259,A -85,B 0,C 180,E1 -14281.622,E2 -14281.622} C_VEL
LIN {X 0,Y 340.005,Z 252.792,A -85,B 0,C 180,E1 -14285.581,E2 -14285.581} C_VEL
LIN {X 0,Y 339.943,Z 255.869,A -85,B 0,C 180,E1 -14288.714,E2 -14288.714} C_VEL
LIN {X 0,Y 343.904,Z 269.049,A -85,B 0,C 180,E1 -14289.526,E2 -14289.526} C_VEL
LIN {X 0,Y 346.943,Z 281.441,A -85,B 0,C 180,E1 -14290.481,E2 -14290.481} C_VEL
LIN {X 0,Y 347.763,Z 285.38,A -85,B 0,C 180,E1 -14290.832,E2 -14290.832} C_VEL
LIN {X 0,Y 346.878,Z 297.281,A -85,B 0,C 180,E1 -14291.85,E2 -14291.85} C_VEL
LIN {X 0,Y 345.827,Z 308.395,A -85,B 0,C 180,E1 -14293.077,E2 -14293.077} C_VEL
LIN {X 0,Y 344.779,Z 317.593,A -85,B 0,C 180,E1 -14294.33,E2 -14294.33} C_VEL
LIN {X 0,Y 343.591,Z 326.4,A -85,B 0,C 180,E1 -14295.791,E2 -14295.791} C_VEL
LIN {X 0,Y 342.426,Z 334.983,A -85,B 0,C 180,E1 -14297.555,E2 -14297.555} C_VEL
LIN {X 0,Y 341.465,Z 341.819,A -85,B 0,C 180,E1 -14299.325,E2 -14299.325} C_VEL
LIN {X 0,Y 340.746,Z 347.286,A -85,B 0,C 180,E1 -14301.101,E2 -14301.101} C_VEL
LIN {X 0,Y 340.237,Z 351.573,A -85,B 0,C 180,E1 -14302.88,E2 -14302.88} C_VEL
LIN {X 0,Y 339.894,Z 353.845,A -85,B 0,C 180,E1 -14304.066,E2 -14304.066} C_VEL
LIN {X 0,Y 339.689,Z 355.689,A -85,B 0,C 180,E1 -14305.253,E2 -14305.253} C_VEL
LIN {X 0,Y 339.651,Z 357.07,A -85,B 0,C 180,E1 -14306.441,E2 -14306.441} C_VEL
LIN {X 0,Y 339.391,Z 358.669,A -85,B 0,C 180,E1 -14308.813,E2 -14308.813} C_VEL
LIN {X 0,Y 339.356,Z 358.9,A -85,B 0,C 180,E1 -14310,E2 -14310} C_VEL
LIN {X 0,Y 339.507,Z 358.126,A -85,B 0,C 180,E1 -14312.373,E2 -14312.373} C_VEL
LIN {X 0,Y 339.631,Z 357.165,A -85,B 0,C 180,E1 -14313.559,E2 -14313.559} C_VEL
LIN {X 0,Y 339.679,Z 355.825,A -85,B 0,C 180,E1 -14314.747,E2 -14314.747} C_VEL
LIN {X 0,Y 340.056,Z 352.976,A -85,B 0,C 180,E1 -14316.527,E2 -14316.527} C_VEL
LIN {X 0,Y 340.51,Z 349.116,A -85,B 0,C 180,E1 -14318.307,E2 -14318.307} C_VEL
LIN {X 0,Y 341.127,Z 344.133,A -85,B 0,C 180,E1 -14320.086,E2 -14320.086} C_VEL
LIN {X 0,Y 342.075,Z 337.846,A -85,B 0,C 180,E1 -14321.856,E2 -14321.856} C_VEL
LIN {X 0,Y 343.163,Z 329.975,A -85,B 0,C 180,E1 -14323.622,E2 -14323.622} C_VEL
LIN {X 0,Y 344.182,Z 321.95,A -85,B 0,C 180,E1 -14325.091,E2 -14325.091} C_VEL
LIN {X 0,Y 345.393,Z 312.147,A -85,B 0,C 180,E1 -14326.551,E2 -14326.551} C_VEL
LIN {X 0,Y 346.382,Z 302.498,A -85,B 0,C 180,E1 -14327.719,E2 -14327.719} C_VEL
LIN {X 0,Y 347.414,Z 292.038,A -85,B 0,C 180,E1 -14328.732,E2 -14328.732} C_VEL
LIN {X 0,Y 347.864,Z 286.181,A -85,B 0,C 180,E1 -14329.206,E2 -14329.206} C_VEL
LIN {X 0,Y 345.53,Z 275.228,A -85,B 0,C 180,E1 -14330.128,E2 -14330.128} C_VEL
LIN {X 0,Y 342.015,Z 262.482,A -85,B 0,C 180,E1 -14331.012,E2 -14331.012} C_VEL
LIN {X 0,Y 339.924,Z 255.741,A -85,B 0,C 180,E1 -14331.415,E2 -14331.415} C_VEL
LIN {X 0,Y 339.992,Z 252.766,A -85,B 0,C 180,E1 -14334.559,E2 -14334.559} C_VEL
LIN {X 0,Y 340.097,Z 249.364,A -85,B 0,C 180,E1 -14338.378,E2 -14338.378} C_VEL
LIN {X 0,Y 340.214,Z 246.214,A -85,B 0,C 180,E1 -14342.117,E2 -14342.117} C_VEL
LIN {X 0,Y 340.553,Z 246.062,A -85,B 0,C 180,E1 -14345.299,E2 -14345.299} C_VEL
LIN {X 0,Y 340.704,Z 246.047,A -85,B 0,C 180,E1 -14348.384,E2 -14348.384} C_VEL
LIN {X 0,Y 340.684,Z 246.047,A -85,B 0,C 180,E1 -14352.322,E2 -14352.322} C_VEL
LIN {X 0,Y 340.654,Z 246.051,A -85,B 0,C 180,E1 -14356.227,E2 -14356.227} C_VEL
LIN {X 0,Y 340.678,Z 246.047,A -85,B 0,C 180,E1 -14357.462,E2 -14357.462} C_VEL
LIN {X 0,Y 340.029,Z 246.132,A -85,B 0,C 180,E1 -14358.449,E2 -14358.449} C_VEL
LIN {X 0,Y 337.179,Z 246.488,A -85,B 0,C 180,E1 -14360.056,E2 -14360.056} C_VEL
LIN {X 0,Y 334.759,Z 246.786,A -85,B 0,C 180,E1 -14361.357,E2 -14361.357} C_VEL
LIN {X 0,Y 333.729,Z 246.913,A -85,B 0,C 180,E1 -14362.364,E2 -14362.364} C_VEL
LIN {X 0,Y 333.651,Z 246.921,A -85,B 0,C 180,E1 -14362.705,E2 -14362.705} C_VEL
LIN {X 0,Y 333.676,Z 246.921,A -85,B 0,C 180,E1 -14365.341,E2 -14365.341} C_VEL
LIN {X 0,Y 333.633,Z 246.924,A -85,B 0,C 180,E1 -14368.222,E2 -14368.222} C_VEL
LIN {X 0,Y 333.656,Z 246.922,A -85,B 0,C 180,E1 -14371.022,E2 -14371.022} C_VEL
LIN {X 0,Y 333.698,Z 246.918,A -85,B 0,C 180,E1 -14375.088,E2 -14375.088} C_VEL
LIN {X 0,Y 333.673,Z 246.921,A -85,B 0,C 180,E1 -14379.019,E2 -14379.019} C_VEL
LIN {X 0,Y 333.743,Z 246.911,A -85,B 0,C 180,E1 -14381.586,E2 -14381.586} C_VEL
LIN {X 0,Y 333.81,Z 246.902,A -85,B 0,C 180,E1 -14385.577,E2 -14385.577} C_VEL
LIN {X 0,Y 333.837,Z 246.902,A -85,B 0,C 180,E1 -14389.078,E2 -14389.078} C_VEL
LIN {X 0,Y 334.027,Z 246.879,A -85,B 0,C 180,E1 -14392.747,E2 -14392.747} C_VEL
LIN {X 0,Y 333.8,Z 246.904,A -85,B 0,C 180,E1 -14395.169,E2 -14395.169} C_VEL
LIN {X 0,Y 334.074,Z 246.868,A -85,B 0,C 180,E1 -14397.589,E2 -14397.589} C_VEL
LIN {X 0,Y 334.085,Z 246.868,A -85,B 0,C 180,E1 -14401.205,E2 -14401.205} C_VEL
LIN {X 0,Y 334.107,Z 246.869,A -85,B 0,C 180,E1 -14402.411,E2 -14402.411} C_VEL
LIN {X 0,Y 334.011,Z 246.879,A -85,B 0,C 180,E1 -14406.039,E2 -14406.039} C_VEL
LIN {X 0,Y 333.821,Z 246.901,A -85,B 0,C 180,E1 -14409.696,E2 -14409.696} C_VEL
LIN {X 0,Y 333.798,Z 246.903,A -85,B 0,C 180,E1 -14413.391,E2 -14413.391} C_VEL
LIN {X 0,Y 333.749,Z 246.909,A -85,B 0,C 180,E1 -14417.146,E2 -14417.146} C_VEL
LIN {X 0,Y 333.737,Z 246.914,A -85,B 0,C 180,E1 -14419.69,E2 -14419.69} C_VEL
LIN {X 0,Y 333.643,Z 246.926,A -85,B 0,C 180,E1 -14423.592,E2 -14423.592} C_VEL
LIN {X 0,Y 333.668,Z 246.925,A -85,B 0,C 180,E1 -14427.606,E2 -14427.606} C_VEL
LIN {X 0,Y 333.659,Z 246.922,A -85,B 0,C 180,E1 -14430.366,E2 -14430.366} C_VEL
LIN {X 0,Y 333.638,Z 246.927,A -85,B 0,C 180,E1 -14433.208,E2 -14433.208} C_VEL
LIN {X 0,Y 333.676,Z 246.919,A -85,B 0,C 180,E1 -14436.139,E2 -14436.139} C_VEL
LIN {X 0,Y 333.621,Z 246.928,A -85,B 0,C 180,E1 -14439.196,E2 -14439.196} C_VEL
LIN {X 0,Y 333.692,Z 247.041,A -85,B 0,C 180,E1 -14441.967,E2 -14441.967} C_VEL
LIN {X 0,Y 334.626,Z 252.003,A -85,B 0,C 180,E1 -14445.569,E2 -14445.569} C_VEL
LIN {X 0,Y 335.7,Z 257.944,A -85,B 0,C 180,E1 -14449.534,E2 -14449.534} C_VEL
LIN {X 0,Y 336.418,Z 263.067,A -85,B 0,C 180,E1 -14452.711,E2 -14452.711} C_VEL
LIN {X 0,Y 336.298,Z 266.306,A -85,B 0,C 180,E1 -14454.59,E2 -14454.59} C_VEL
LIN {X 0,Y 335.374,Z 273.222,A -85,B 0,C 180,E1 -14458.406,E2 -14458.406} C_VEL
LIN {X 0,Y 334.449,Z 280.743,A -85,B 0,C 180,E1 -14462.464,E2 -14462.464} C_VEL
LIN {X 0,Y 333.773,Z 286.937,A -85,B 0,C 180,E1 -14465.758,E2 -14465.758} C_VEL
LIN {X 0,Y 333.378,Z 291.43,A -85,B 0,C 180,E1 -14468.148,E2 -14468.148} C_VEL
LIN {X 0,Y 335.952,Z 305.098,A -85,B 0,C 180,E1 -14468.841,E2 -14468.841} C_VEL
LIN {X 0,Y 337.68,Z 317.84,A -85,B 0,C 180,E1 -14469.696,E2 -14469.696} C_VEL
LIN {X 0,Y 338.673,Z 328.781,A -85,B 0,C 180,E1 -14470.608,E2 -14470.608} C_VEL
LIN {X 0,Y 339.102,Z 333.89,A -85,B 0,C 180,E1 -14471.105,E2 -14471.105} C_VEL
LIN {X 0,Y 337.774,Z 345.221,A -85,B 0,C 180,E1 -14472.284,E2 -14472.284} C_VEL
LIN {X 0,Y 336.479,Z 355.447,A -85,B 0,C 180,E1 -14473.623,E2 -14473.623} C_VEL
LIN {X 0,Y 335.382,Z 364.789,A -85,B 0,C 180,E1 -14475.15,E2 -14475.15} C_VEL
LIN {X 0,Y 334.252,Z 373.648,A -85,B 0,C 180,E1 -14476.937,E2 -14476.937} C_VEL
LIN {X 0,Y 333.323,Z 380.887,A -85,B 0,C 180,E1 -14478.753,E2 -14478.753} C_VEL
LIN {X 0,Y 332.819,Z 385.784,A -85,B 0,C 180,E1 -14480.274,E2 -14480.274} C_VEL
LIN {X 0,Y 332.389,Z 390.549,A -85,B 0,C 180,E1 -14482.101,E2 -14482.101} C_VEL
LIN {X 0,Y 332.181,Z 394.197,A -85,B 0,C 180,E1 -14483.928,E2 -14483.928} C_VEL
LIN {X 0,Y 332.116,Z 396.082,A -85,B 0,C 180,E1 -14485.145,E2 -14485.145} C_VEL
LIN {X 0,Y 332.057,Z 397.494,A -85,B 0,C 180,E1 -14486.36,E2 -14486.36} C_VEL
LIN {X 0,Y 332.133,Z 399.126,A -85,B 0,C 180,E1 -14488.788,E2 -14488.788} C_VEL
LIN {X 0,Y 332.213,Z 399.349,A -85,B 0,C 180,E1 -14490,E2 -14490} C_VEL
LIN {X 0,Y 332.133,Z 399.123,A -85,B 0,C 180,E1 -14491.213,E2 -14491.213} C_VEL
LIN {X 0,Y 332.057,Z 397.49,A -85,B 0,C 180,E1 -14493.641,E2 -14493.641} C_VEL
LIN {X 0,Y 332.115,Z 396.075,A -85,B 0,C 180,E1 -14494.856,E2 -14494.856} C_VEL
LIN {X 0,Y 332.219,Z 393.099,A -85,B 0,C 180,E1 -14496.682,E2 -14496.682} C_VEL
LIN {X 0,Y 332.493,Z 389.08,A -85,B 0,C 180,E1 -14498.509,E2 -14498.509} C_VEL
LIN {X 0,Y 333.13,Z 382.914,A -85,B 0,C 180,E1 -14500.638,E2 -14500.638} C_VEL
LIN {X 0,Y 333.907,Z 376.186,A -85,B 0,C 180,E1 -14502.459,E2 -14502.459} C_VEL
LIN {X 0,Y 334.947,Z 367.85,A -85,B 0,C 180,E1 -14504.273,E2 -14504.273} C_VEL
LIN {X 0,Y 336.146,Z 358.524,A -85,B 0,C 180,E1 -14505.898,E2 -14505.898} C_VEL
LIN {X 0,Y 337.404,Z 347.591,A -85,B 0,C 180,E1 -14507.423,E2 -14507.423} C_VEL
LIN {X 0,Y 338.796,Z 336.933,A -85,B 0,C 180,E1 -14508.599,E2 -14508.599} C_VEL
LIN {X 0,Y 339.015,Z 332.188,A -85,B 0,C 180,E1 -14509.057,E2 -14509.057} C_VEL
LIN {X 0,Y 337.932,Z 319.76,A -85,B 0,C 180,E1 -14510.145,E2 -14510.145} C_VEL
LIN {X 0,Y 336.141,Z 306.304,A -85,B 0,C 180,E1 -14511.073,E2 -14511.073} C_VEL
LIN {X 0,Y 333.655,Z 293.258,A -85,B 0,C 180,E1 -14511.768,E2 -14511.768} C_VEL
LIN {X 0,Y 333.378,Z 291.349,A -85,B 0,C 180,E1 -14511.853,E2 -14511.853} C_VEL
LIN {X 0,Y 333.984,Z 285.12,A -85,B 0,C 180,E1 -14515.197,E2 -14515.197} C_VEL
LIN {X 0,Y 334.731,Z 278.226,A -85,B 0,C 180,E1 -14518.876,E2 -14518.876} C_VEL
LIN {X 0,Y 335.745,Z 270.338,A -85,B 0,C 180,E1 -14523.143,E2 -14523.143} C_VEL
LIN {X 0,Y 336.476,Z 264.245,A -85,B 0,C 180,E1 -14526.533,E2 -14526.533} C_VEL
LIN {X 0,Y 335.988,Z 259.688,A -85,B 0,C 180,E1 -14529.29,E2 -14529.29} C_VEL
LIN {X 0,Y 335.048,Z 254.355,A -85,B 0,C 180,E1 -14532.763,E2 -14532.763} C_VEL
LIN {X 0,Y 334.182,Z 249.672,A -85,B 0,C 180,E1 -14536.052,E2 -14536.052} C_VEL
LIN {X 0,Y 333.655,Z 246.925,A -85,B 0,C 180,E1 -14538.23,E2 -14538.23} C_VEL
LIN {X 0,Y 333.646,Z 246.926,A -85,B 0,C 180,E1 -14542.348,E2 -14542.348} C_VEL
LIN {X 0,Y 333.677,Z 246.919,A -85,B 0,C 180,E1 -14545.342,E2 -14545.342} C_VEL
LIN {X 0,Y 333.633,Z 246.927,A -85,B 0,C 180,E1 -14548.222,E2 -14548.222} C_VEL
LIN {X 0,Y 333.657,Z 246.921,A -85,B 0,C 180,E1 -14551.023,E2 -14551.023} C_VEL
LIN {X 0,Y 333.667,Z 246.92,A -85,B 0,C 180,E1 -14555.086,E2 -14555.086} C_VEL
LIN {X 0,Y 333.67,Z 246.92,A -85,B 0,C 180,E1 -14559.019,E2 -14559.019} C_VEL
LIN {X 0,Y 333.798,Z 246.905,A -85,B 0,C 180,E1 -14561.59,E2 -14561.59} C_VEL
LIN {X 0,Y 333.812,Z 246.904,A -85,B 0,C 180,E1 -14565.577,E2 -14565.577} C_VEL
LIN {X 0,Y 333.818,Z 246.901,A -85,B 0,C 180,E1 -14569.078,E2 -14569.078} C_VEL
LIN {X 0,Y 333.996,Z 246.878,A -85,B 0,C 180,E1 -14572.747,E2 -14572.747} C_VEL
LIN {X 0,Y 333.81,Z 246.903,A -85,B 0,C 180,E1 -14575.169,E2 -14575.169} C_VEL
LIN {X 0,Y 334.109,Z 246.869,A -85,B 0,C 180,E1 -14577.589,E2 -14577.589} C_VEL
LIN {X 0,Y 334.063,Z 246.873,A -85,B 0,C 180,E1 -14581.206,E2 -14581.206} C_VEL
LIN {X 0,Y 334.075,Z 246.868,A -85,B 0,C 180,E1 -14582.411,E2 -14582.411} C_VEL
LIN {X 0,Y 333.985,Z 246.88,A -85,B 0,C 180,E1 -14586.635,E2 -14586.635} C_VEL
LIN {X 0,Y 333.825,Z 246.901,A -85,B 0,C 180,E1 -14589.696,E2 -14589.696} C_VEL
LIN {X 0,Y 333.801,Z 246.905,A -85,B 0,C 180,E1 -14593.391,E2 -14593.391} C_VEL
LIN {X 0,Y 333.723,Z 246.915,A -85,B 0,C 180,E1 -14597.148,E2 -14597.148} C_VEL
LIN {X 0,Y 333.689,Z 246.917,A -85,B 0,C 180,E1 -14599.693,E2 -14599.693} C_VEL
LIN {X 0,Y 333.664,Z 246.919,A -85,B 0,C 180,E1 -14603.591,E2 -14603.591} C_VEL
LIN {X 0,Y 333.662,Z 246.922,A -85,B 0,C 180,E1 -14606.253,E2 -14606.253} C_VEL
LIN {X 0,Y 333.664,Z 246.923,A -85,B 0,C 180,E1 -14610.277,E2 -14610.277} C_VEL
LIN {X 0,Y 333.64,Z 246.923,A -85,B 0,C 180,E1 -14613.208,E2 -14613.208} C_VEL
LIN {X 0,Y 333.679,Z 246.921,A -85,B 0,C 180,E1 -14616.139,E2 -14616.139} C_VEL
LIN {X 0,Y 333.65,Z 246.921,A -85,B 0,C 180,E1 -14619.192,E2 -14619.192} C_VEL
LIN {X 0,Y 333.635,Z 246.926,A -85,B 0,C 180,E1 -14622.5,E2 -14622.5} C_VEL
LIN {X 0,Y 333.599,Z 246.932,A -85,B 0,C 180,E1 -14625.955,E2 -14625.955} C_VEL
LIN {X 0,Y 333.649,Z 246.923,A -85,B 0,C 180,E1 -14629.315,E2 -14629.315} C_VEL
LIN {X 0,Y 333.634,Z 246.924,A -85,B 0,C 180,E1 -14633.175,E2 -14633.175} C_VEL
LIN {X 0,Y 333.476,Z 246.945,A -85,B 0,C 180,E1 -14635.317,E2 -14635.317} C_VEL
LIN {X 0,Y 333.2,Z 246.983,A -85,B 0,C 180,E1 -14637.533,E2 -14637.533} C_VEL
LIN {X 0,Y 333.083,Z 249.648,A -85,B 0,C 180,E1 -14640.968,E2 -14640.968} C_VEL
LIN {X 0,Y 332.956,Z 253.205,A -85,B 0,C 180,E1 -14645.029,E2 -14645.029} C_VEL
LIN {X 0,Y 332.903,Z 256.227,A -85,B 0,C 180,E1 -14648.23,E2 -14648.23} C_VEL
LIN {X 0,Y 337.12,Z 270.242,A -85,B 0,C 180,E1 -14649.134,E2 -14649.134} C_VEL
LIN {X 0,Y 340.149,Z 282.518,A -85,B 0,C 180,E1 -14650.12,E2 -14650.12} C_VEL
LIN {X 0,Y 341.003,Z 287.883,A -85,B 0,C 180,E1 -14650.602,E2 -14650.602} C_VEL
LIN {X 0,Y 340.025,Z 299.147,A -85,B 0,C 180,E1 -14651.627,E2 -14651.627} C_VEL
LIN {X 0,Y 338.942,Z 310.062,A -85,B 0,C 180,E1 -14652.888,E2 -14652.888} C_VEL
LIN {X 0,Y 337.711,Z 319.959,A -85,B 0,C 180,E1 -14654.303,E2 -14654.303} C_VEL
LIN {X 0,Y 336.567,Z 328.417,A -85,B 0,C 180,E1 -14655.797,E2 -14655.797} C_VEL
LIN {X 0,Y 335.323,Z 336.633,A -85,B 0,C 180,E1 -14657.594,E2 -14657.594} C_VEL
LIN {X 0,Y 334.494,Z 342.249,A -85,B 0,C 180,E1 -14659.1,E2 -14659.1} C_VEL
LIN {X 0,Y 333.759,Z 347.714,A -85,B 0,C 180,E1 -14660.913,E2 -14660.913} C_VEL
LIN {X 0,Y 333.191,Z 352.002,A -85,B 0,C 180,E1 -14662.729,E2 -14662.729} C_VEL
LIN {X 0,Y 332.865,Z 354.272,A -85,B 0,C 180,E1 -14663.94,E2 -14663.94} C_VEL
LIN {X 0,Y 332.624,Z 356.117,A -85,B 0,C 180,E1 -14665.152,E2 -14665.152} C_VEL
LIN {X 0,Y 332.568,Z 357.498,A -85,B 0,C 180,E1 -14666.365,E2 -14666.365} C_VEL
LIN {X 0,Y 332.333,Z 359.094,A -85,B 0,C 180,E1 -14668.788,E2 -14668.788} C_VEL
LIN {X 0,Y 332.296,Z 359.325,A -85,B 0,C 180,E1 -14670,E2 -14670} C_VEL
LIN {X 0,Y 332.333,Z 359.135,A -85,B 0,C 180,E1 -14671.212,E2 -14671.212} C_VEL
LIN {X 0,Y 332.549,Z 357.592,A -85,B 0,C 180,E1 -14673.635,E2 -14673.635} C_VEL
LIN {X 0,Y 332.614,Z 356.251,A -85,B 0,C 180,E1 -14674.848,E2 -14674.848} C_VEL
LIN {X 0,Y 333.028,Z 353.401,A -85,B 0,C 180,E1 -14676.665,E2 -14676.665} C_VEL
LIN {X 0,Y 333.504,Z 349.542,A -85,B 0,C 180,E1 -14678.483,E2 -14678.483} C_VEL
LIN {X 0,Y 334.16,Z 344.558,A -85,B 0,C 180,E1 -14680.298,E2 -14680.298} C_VEL
LIN {X 0,Y 335.142,Z 338.27,A -85,B 0,C 180,E1 -14682.105,E2 -14682.105} C_VEL
LIN {X 0,Y 336.291,Z 330.399,A -85,B 0,C 180,E1 -14683.906,E2 -14683.906} C_VEL
LIN {X 0,Y 337.354,Z 322.373,A -85,B 0,C 180,E1 -14685.404,E2 -14685.404} C_VEL
LIN {X 0,Y 338.62,Z 312.569,A -85,B 0,C 180,E1 -14686.892,E2 -14686.892} C_VEL
LIN {X 0,Y 339.638,Z 302.92,A -85,B 0,C 180,E1 -14688.083,E2 -14688.083} C_VEL
LIN {X 0,Y 340.722,Z 292.458,A -85,B 0,C 180,E1 -14689.114,E2 -14689.114} C_VEL
LIN {X 0,Y 341.085,Z 286.895,A -85,B 0,C 180,E1 -14689.58,E2 -14689.58} C_VEL
LIN {X 0,Y 338.614,Z 275.656,A -85,B 0,C 180,E1 -14690.558,E2 -14690.558} C_VEL
LIN {X 0,Y 334.914,Z 262.665,A -85,B 0,C 180,E1 -14691.491,E2 -14691.491} C_VEL
LIN {X 0,Y 332.892,Z 256.182,A -85,B 0,C 180,E1 -14691.877,E2 -14691.877} C_VEL
LIN {X 0,Y 332.933,Z 253.308,A -85,B 0,C 180,E1 -14694.973,E2 -14694.973} C_VEL
LIN {X 0,Y 333.079,Z 249.759,A -85,B 0,C 180,E1 -14699.032,E2 -14699.032} C_VEL
LIN {X 0,Y 333.195,Z 246.987,A -85,B 0,C 180,E1 -14702.466,E2 -14702.466} C_VEL
LIN {X 0,Y 333.47,Z 246.947,A -85,B 0,C 180,E1 -14704.72,E2 -14704.72} C_VEL
LIN {X 0,Y 333.636,Z 246.926,A -85,B 0,C 180,E1 -14707.653,E2 -14707.653} C_VEL
LIN {X 0,Y 333.648,Z 246.923,A -85,B 0,C 180,E1 -14710.767,E2 -14710.767} C_VEL
LIN {X 0,Y 333.595,Z 246.932,A -85,B 0,C 180,E1 -14714.25,E2 -14714.25} C_VEL
LIN {X 0,Y 333.643,Z 246.924,A -85,B 0,C 180,E1 -14717.618,E2 -14717.618} C_VEL
LIN {X 0,Y 333.654,Z 246.922,A -85,B 0,C 180,E1 -14721.202,E2 -14721.202} C_VEL
LIN {X 0,Y 333.651,Z 246.921,A -85,B 0,C 180,E1 -14722.705,E2 -14722.705} C_VEL
LIN {X 0,Y 332.999,Z 247.007,A -85,B 0,C 180,E1 -14723.712,E2 -14723.712} C_VEL
LIN {X 0,Y 330.154,Z 247.36,A -85,B 0,C 180,E1 -14725.352,E2 -14725.352} C_VEL
LIN {X 0,Y 327.723,Z 247.663,A -85,B 0,C 180,E1 -14726.68,E2 -14726.68} C_VEL
LIN {X 0,Y 326.665,Z 247.795,A -85,B 0,C 180,E1 -14727.708,E2 -14727.708} C_VEL
LIN {X 0,Y 326.572,Z 247.802,A -85,B 0,C 180,E1 -14728.057,E2 -14728.057} C_VEL
LIN {X 0,Y 326.6,Z 247.802,A -85,B 0,C 180,E1 -14731.744,E2 -14731.744} C_VEL
LIN {X 0,Y 326.643,Z 247.794,A -85,B 0,C 180,E1 -14734.644,E2 -14734.644} C_VEL
LIN {X 0,Y 326.62,Z 247.797,A -85,B 0,C 180,E1 -14738.543,E2 -14738.543} C_VEL
LIN {X 0,Y 326.709,Z 247.79,A -85,B 0,C 180,E1 -14741.175,E2 -14741.175} C_VEL
LIN {X 0,Y 326.765,Z 247.781,A -85,B 0,C 180,E1 -14745.433,E2 -14745.433} C_VEL
LIN {X 0,Y 326.773,Z 247.782,A -85,B 0,C 180,E1 -14748.839,E2 -14748.839} C_VEL
LIN {X 0,Y 326.981,Z 247.755,A -85,B 0,C 180,E1 -14752.59,E2 -14752.59} C_VEL
LIN {X 0,Y 326.769,Z 247.781,A -85,B 0,C 180,E1 -14755.065,E2 -14755.065} C_VEL
LIN {X 0,Y 327.018,Z 247.748,A -85,B 0,C 180,E1 -14757.536,E2 -14757.536} C_VEL
LIN {X 0,Y 327.054,Z 247.744,A -85,B 0,C 180,E1 -14761.231,E2 -14761.231} C_VEL
LIN {X 0,Y 327.048,Z 247.749,A -85,B 0,C 180,E1 -14762.463,E2 -14762.463} C_VEL
LIN {X 0,Y 326.985,Z 247.755,A -85,B 0,C 180,E1 -14766.169,E2 -14766.169} C_VEL
LIN {X 0,Y 326.784,Z 247.779,A -85,B 0,C 180,E1 -14769.907,E2 -14769.907} C_VEL
LIN {X 0,Y 326.76,Z 247.781,A -85,B 0,C 180,E1 -14773.685,E2 -14773.685} C_VEL
LIN {X 0,Y 326.702,Z 247.788,A -85,B 0,C 180,E1 -14777.528,E2 -14777.528} C_VEL
LIN {X 0,Y 326.66,Z 247.796,A -85,B 0,C 180,E1 -14780.135,E2 -14780.135} C_VEL
LIN {X 0,Y 326.611,Z 247.802,A -85,B 0,C 180,E1 -14784.132,E2 -14784.132} C_VEL
LIN {X 0,Y 326.6,Z 247.803,A -85,B 0,C 180,E1 -14788.256,E2 -14788.256} C_VEL
LIN {X 0,Y 326.575,Z 247.806,A -85,B 0,C 180,E1 -14791.097,E2 -14791.097} C_VEL
LIN {X 0,Y 326.608,Z 247.802,A -85,B 0,C 180,E1 -14794.019,E2 -14794.019} C_VEL
LIN {X 0,Y 326.624,Z 247.802,A -85,B 0,C 180,E1 -14797.237,E2 -14797.237} C_VEL
LIN {X 0,Y 326.624,Z 247.898,A -85,B 0,C 180,E1 -14801.428,E2 -14801.428} C_VEL
LIN {X 0,Y 327.55,Z 252.765,A -85,B 0,C 180,E1 -14805.077,E2 -14805.077} C_VEL
LIN {X 0,Y 328.681,Z 258.942,A -85,B 0,C 180,E1 -14809.316,E2 -14809.316} C_VEL
LIN {X 0,Y 329.363,Z 263.338,A -85,B 0,C 180,E1 -14812.14,E2 -14812.14} C_VEL
LIN {X 0,Y 329.364,Z 266.74,A -85,B 0,C 180,E1 -14814.179,E2 -14814.179} C_VEL
LIN {X 0,Y 328.484,Z 272.864,A -85,B 0,C 180,E1 -14817.664,E2 -14817.664} C_VEL
LIN {X 0,Y 327.586,Z 279.937,A -85,B 0,C 180,E1 -14821.596,E2 -14821.596} C_VEL
LIN {X 0,Y 326.809,Z 286.515,A -85,B 0,C 180,E1 -14825.207,E2 -14825.207} C_VEL
LIN {X 0,Y 326.381,Z 291.085,A -85,B 0,C 180,E1 -14827.662,E2 -14827.662} C_VEL
LIN {X 0,Y 328.984,Z 304.453,A -85,B 0,C 180,E1 -14828.36,E2 -14828.36} C_VEL
LIN {X 0,Y 330.744,Z 316.992,A -85,B 0,C 180,E1 -14829.222,E2 -14829.222} C_VEL
LIN {X 0,Y 331.782,Z 328.346,A -85,B 0,C 180,E1 -14830.189,E2 -14830.189} C_VEL
LIN {X 0,Y 332.207,Z 335.055,A -85,B 0,C 180,E1 -14830.858,E2 -14830.858} C_VEL
LIN {X 0,Y 330.817,Z 346.059,A -85,B 0,C 180,E1 -14832.059,E2 -14832.059} C_VEL
LIN {X 0,Y 329.621,Z 355.015,A -85,B 0,C 180,E1 -14833.271,E2 -14833.271} C_VEL
LIN {X 0,Y 328.475,Z 364.544,A -85,B 0,C 180,E1 -14834.865,E2 -14834.865} C_VEL
LIN {X 0,Y 327.315,Z 373.221,A -85,B 0,C 180,E1 -14836.655,E2 -14836.655} C_VEL
LIN {X 0,Y 326.299,Z 380.457,A -85,B 0,C 180,E1 -14838.508,E2 -14838.508} C_VEL
LIN {X 0,Y 325.803,Z 385.356,A -85,B 0,C 180,E1 -14840.063,E2 -14840.063} C_VEL
LIN {X 0,Y 325.333,Z 390.121,A -85,B 0,C 180,E1 -14841.928,E2 -14841.928} C_VEL
LIN {X 0,Y 325.103,Z 394.031,A -85,B 0,C 180,E1 -14843.945,E2 -14843.945} C_VEL
LIN {X 0,Y 324.986,Z 397.068,A -85,B 0,C 180,E1 -14846.28,E2 -14846.28} C_VEL
LIN {X 0,Y 325.04,Z 398.699,A -85,B 0,C 180,E1 -14848.761,E2 -14848.761} C_VEL
LIN {X 0,Y 325.138,Z 398.923,A -85,B 0,C 180,E1 -14850,E2 -14850} C_VEL
LIN {X 0,Y 325.04,Z 398.696,A -85,B 0,C 180,E1 -14851.239,E2 -14851.239} C_VEL
LIN {X 0,Y 324.986,Z 397.063,A -85,B 0,C 180,E1 -14853.72,E2 -14853.72} C_VEL
LIN {X 0,Y 325.083,Z 394.075,A -85,B 0,C 180,E1 -14856.023,E2 -14856.023} C_VEL
LIN {X 0,Y 325.301,Z 390.096,A -85,B 0,C 180,E1 -14858.073,E2 -14858.073} C_VEL
LIN {X 0,Y 325.803,Z 385.328,A -85,B 0,C 180,E1 -14859.938,E2 -14859.938} C_VEL
LIN {X 0,Y 326.571,Z 378.168,A -85,B 0,C 180,E1 -14862.112,E2 -14862.112} C_VEL
LIN {X 0,Y 327.698,Z 370.42,A -85,B 0,C 180,E1 -14863.962,E2 -14863.962} C_VEL
LIN {X 0,Y 328.885,Z 361.684,A -85,B 0,C 180,E1 -14865.636,E2 -14865.636} C_VEL
LIN {X 0,Y 330.019,Z 351.741,A -85,B 0,C 180,E1 -14867.187,E2 -14867.187} C_VEL
LIN {X 0,Y 331.474,Z 340.79,A -85,B 0,C 180,E1 -14868.544,E2 -14868.544} C_VEL
LIN {X 0,Y 332.176,Z 333.347,A -85,B 0,C 180,E1 -14869.305,E2 -14869.305} C_VEL
LIN {X 0,Y 331.257,Z 321.847,A -85,B 0,C 180,E1 -14870.378,E2 -14870.378} C_VEL
LIN {X 0,Y 329.63,Z 308.782,A -85,B 0,C 180,E1 -14871.354,E2 -14871.354} C_VEL
LIN {X 0,Y 327.389,Z 296.034,A -85,B 0,C 180,E1 -14872.092,E2 -14872.092} C_VEL
LIN {X 0,Y 326.395,Z 290.959,A -85,B 0,C 180,E1 -14872.33,E2 -14872.33} C_VEL
LIN {X 0,Y 327.077,Z 284.053,A -85,B 0,C 180,E1 -14876.135,E2 -14876.135} C_VEL
LIN {X 0,Y 327.826,Z 277.848,A -85,B 0,C 180,E1 -14879.544,E2 -14879.544} C_VEL
LIN {X 0,Y 328.879,Z 270.283,A -85,B 0,C 180,E1 -14883.753,E2 -14883.753} C_VEL
LIN {X 0,Y 329.472,Z 265.179,A -85,B 0,C 180,E1 -14886.675,E2 -14886.675} C_VEL
LIN {X 0,Y 329.09,Z 261.452,A -85,B 0,C 180,E1 -14888.973,E2 -14888.973} C_VEL
LIN {X 0,Y 328.193,Z 256.291,A -85,B 0,C 180,E1 -14892.401,E2 -14892.401} C_VEL
LIN {X 0,Y 327.289,Z 251.44,A -85,B 0,C 180,E1 -14895.832,E2 -14895.832} C_VEL
LIN {X 0,Y 326.582,Z 247.806,A -85,B 0,C 180,E1 -14898.769,E2 -14898.769} C_VEL
LIN {X 0,Y 326.626,Z 247.801,A -85,B 0,C 180,E1 -14902.763,E2 -14902.763} C_VEL
LIN {X 0,Y 326.61,Z 247.8,A -85,B 0,C 180,E1 -14905.981,E2 -14905.981} C_VEL
LIN {X 0,Y 326.615,Z 247.798,A -85,B 0,C 180,E1 -14909.397,E2 -14909.397} C_VEL
LIN {X 0,Y 326.605,Z 247.8,A -85,B 0,C 180,E1 -14913.135,E2 -14913.135} C_VEL
LIN {X 0,Y 326.594,Z 247.801,A -85,B 0,C 180,E1 -14917.211,E2 -14917.211} C_VEL
LIN {X 0,Y 326.748,Z 247.782,A -85,B 0,C 180,E1 -14921.178,E2 -14921.178} C_VEL
LIN {X 0,Y 326.767,Z 247.781,A -85,B 0,C 180,E1 -14925.433,E2 -14925.433} C_VEL
LIN {X 0,Y 326.759,Z 247.78,A -85,B 0,C 180,E1 -14928.839,E2 -14928.839} C_VEL
LIN {X 0,Y 326.946,Z 247.756,A -85,B 0,C 180,E1 -14932.59,E2 -14932.59} C_VEL
LIN {X 0,Y 326.986,Z 247.756,A -85,B 0,C 180,E1 -14933.831,E2 -14933.831} C_VEL
LIN {X 0,Y 327.05,Z 247.749,A -85,B 0,C 180,E1 -14937.537,E2 -14937.537} C_VEL
LIN {X 0,Y 327.033,Z 247.749,A -85,B 0,C 180,E1 -14941.231,E2 -14941.231} C_VEL
LIN {X 0,Y 326.769,Z 247.781,A -85,B 0,C 180,E1 -14943.7,E2 -14943.7} C_VEL
LIN {X 0,Y 326.941,Z 247.756,A -85,B 0,C 180,E1 -14946.628,E2 -14946.628} C_VEL
LIN {X 0,Y 326.787,Z 247.777,A -85,B 0,C 180,E1 -14949.907,E2 -14949.907} C_VEL
LIN {X 0,Y 326.763,Z 247.78,A -85,B 0,C 180,E1 -14953.685,E2 -14953.685} C_VEL
LIN {X 0,Y 326.667,Z 247.791,A -85,B 0,C 180,E1 -14957.53,E2 -14957.53} C_VEL
LIN {X 0,Y 326.635,Z 247.796,A -85,B 0,C 180,E1 -14960.137,E2 -14960.137} C_VEL
LIN {X 0,Y 326.637,Z 247.796,A -85,B 0,C 180,E1 -14964.13,E2 -14964.13} C_VEL
LIN {X 0,Y 326.606,Z 247.8,A -85,B 0,C 180,E1 -14968.084,E2 -14968.084} C_VEL
LIN {X 0,Y 326.576,Z 247.804,A -85,B 0,C 180,E1 -14971.097,E2 -14971.097} C_VEL
LIN {X 0,Y 326.61,Z 247.8,A -85,B 0,C 180,E1 -14974.019,E2 -14974.019} C_VEL
LIN {X 0,Y 326.631,Z 247.796,A -85,B 0,C 180,E1 -14977.238,E2 -14977.238} C_VEL
LIN {X 0,Y 326.581,Z 247.802,A -85,B 0,C 180,E1 -14981.131,E2 -14981.131} C_VEL
LIN {X 0,Y 326.53,Z 247.809,A -85,B 0,C 180,E1 -14984.743,E2 -14984.743} C_VEL
LIN {X 0,Y 326.578,Z 247.807,A -85,B 0,C 180,E1 -14988.154,E2 -14988.154} C_VEL
LIN {X 0,Y 326.595,Z 247.802,A -85,B 0,C 180,E1 -14991.387,E2 -14991.387} C_VEL
LIN {X 0,Y 326.459,Z 247.818,A -85,B 0,C 180,E1 -14994.461,E2 -14994.461} C_VEL
LIN {X 0,Y 326.165,Z 247.859,A -85,B 0,C 180,E1 -14997.405,E2 -14997.405} C_VEL
LIN {X 0,Y 326.051,Z 250.04,A -85,B 0,C 180,E1 -15000.279,E2 -15000.279} C_VEL
LIN {X 0,Y 325.951,Z 252.418,A -85,B 0,C 180,E1 -15003.077,E2 -15003.077} C_VEL
LIN {X 0,Y 325.869,Z 254.866,A -85,B 0,C 180,E1 -15005.809,E2 -15005.809} C_VEL
LIN {X 0,Y 325.84,Z 256.666,A -85,B 0,C 180,E1 -15007.733,E2 -15007.733} C_VEL
LIN {X 0,Y 330.123,Z 270.509,A -85,B 0,C 180,E1 -15008.66,E2 -15008.66} C_VEL
LIN {X 0,Y 333.133,Z 282.355,A -85,B 0,C 180,E1 -15009.638,E2 -15009.638} C_VEL
LIN {X 0,Y 334.259,Z 288.457,A -85,B 0,C 180,E1 -15010.207,E2 -15010.207} C_VEL
LIN {X 0,Y 333.301,Z 299.579,A -85,B 0,C 180,E1 -15011.242,E2 -15011.242} C_VEL
LIN {X 0,Y 332.153,Z 310.657,A -85,B 0,C 180,E1 -15012.549,E2 -15012.549} C_VEL
LIN {X 0,Y 330.905,Z 320.389,A -85,B 0,C 180,E1 -15013.972,E2 -15013.972} C_VEL
LIN {X 0,Y 329.7,Z 328.846,A -85,B 0,C 180,E1 -15015.495,E2 -15015.495} C_VEL
LIN {X 0,Y 328.408,Z 337.062,A -85,B 0,C 180,E1 -15017.329,E2 -15017.329} C_VEL
LIN {X 0,Y 327.545,Z 342.677,A -85,B 0,C 180,E1 -15018.865,E2 -15018.865} C_VEL
LIN {X 0,Y 326.752,Z 348.143,A -85,B 0,C 180,E1 -15020.717,E2 -15020.717} C_VEL
LIN {X 0,Y 326.156,Z 352.431,A -85,B 0,C 180,E1 -15022.571,E2 -15022.571} C_VEL
LIN {X 0,Y 325.839,Z 354.699,A -85,B 0,C 180,E1 -15023.809,E2 -15023.809} C_VEL
LIN {X 0,Y 325.564,Z 356.545,A -85,B 0,C 180,E1 -15025.046,E2 -15025.046} C_VEL
LIN {X 0,Y 325.487,Z 357.926,A -85,B 0,C 180,E1 -15026.286,E2 -15026.286} C_VEL
LIN {X 0,Y 325.372,Z 358.911,A -85,B 0,C 180,E1 -15027.524,E2 -15027.524} C_VEL
LIN {X 0,Y 325.236,Z 359.751,A -85,B 0,C 180,E1 -15030,E2 -15030} C_VEL
LIN {X 0,Y 325.368,Z 358.977,A -85,B 0,C 180,E1 -15032.476,E2 -15032.476} C_VEL
LIN {X 0,Y 325.467,Z 358.019,A -85,B 0,C 180,E1 -15033.714,E2 -15033.714} C_VEL
LIN {X 0,Y 325.554,Z 356.677,A -85,B 0,C 180,E1 -15034.954,E2 -15034.954} C_VEL
LIN {X 0,Y 326.026,Z 353.368,A -85,B 0,C 180,E1 -15037.062,E2 -15037.062} C_VEL
LIN {X 0,Y 326.702,Z 348.42,A -85,B 0,C 180,E1 -15039.285,E2 -15039.285} C_VEL
LIN {X 0,Y 327.689,Z 342.017,A -85,B 0,C 180,E1 -15041.443,E2 -15041.443} C_VEL
LIN {X 0,Y 328.723,Z 334.978,A -85,B 0,C 180,E1 -15043.287,E2 -15043.287} C_VEL
LIN {X 0,Y 330.063,Z 326.196,A -85,B 0,C 180,E1 -15045.12,E2 -15045.12} C_VEL
LIN {X 0,Y 331.374,Z 317.177,A -85,B 0,C 180,E1 -15046.638,E2 -15046.638} C_VEL
LIN {X 0,Y 332.516,Z 306.964,A -85,B 0,C 180,E1 -15048.034,E2 -15048.034} C_VEL
LIN {X 0,Y 333.742,Z 296.067,A -85,B 0,C 180,E1 -15049.21,E2 -15049.21} C_VEL
LIN {X 0,Y 334.345,Z 289.407,A -85,B 0,C 180,E1 -15049.809,E2 -15049.809} C_VEL
LIN {X 0,Y 332.973,Z 281.682,A -85,B 0,C 180,E1 -15050.531,E2 -15050.531} C_VEL
LIN {X 0,Y 329.806,Z 269.347,A -85,B 0,C 180,E1 -15051.536,E2 -15051.536} C_VEL
LIN {X 0,Y 325.847,Z 256.611,A -85,B 0,C 180,E1 -15052.379,E2 -15052.379} C_VEL
LIN {X 0,Y 325.896,Z 253.723,A -85,B 0,C 180,E1 -15055.55,E2 -15055.55} C_VEL
LIN {X 0,Y 325.995,Z 251.331,A -85,B 0,C 180,E1 -15058.313,E2 -15058.313} C_VEL
LIN {X 0,Y 326.1,Z 248.978,A -85,B 0,C 180,E1 -15061.147,E2 -15061.147} C_VEL
LIN {X 0,Y 326.181,Z 247.86,A -85,B 0,C 180,E1 -15062.827,E2 -15062.827} C_VEL
LIN {X 0,Y 326.458,Z 247.819,A -85,B 0,C 180,E1 -15065.539,E2 -15065.539} C_VEL
LIN {X 0,Y 326.594,Z 247.804,A -85,B 0,C 180,E1 -15068.613,E2 -15068.613} C_VEL
LIN {X 0,Y 326.577,Z 247.806,A -85,B 0,C 180,E1 -15071.846,E2 -15071.846} C_VEL
LIN {X 0,Y 326.529,Z 247.809,A -85,B 0,C 180,E1 -15075.257,E2 -15075.257} C_VEL
LIN {X 0,Y 326.579,Z 247.802,A -85,B 0,C 180,E1 -15078.869,E2 -15078.869} C_VEL
LIN {X 0,Y 326.629,Z 247.796,A -85,B 0,C 180,E1 -15082.761,E2 -15082.761} C_VEL
LIN {X 0,Y 326.61,Z 247.801,A -85,B 0,C 180,E1 -15085.981,E2 -15085.981} C_VEL
LIN {X 0,Y 326.572,Z 247.802,A -85,B 0,C 180,E1 -15088.057,E2 -15088.057} C_VEL
LIN {X 0,Y 325.879,Z 247.892,A -85,B 0,C 180,E1 -15089.087,E2 -15089.087} C_VEL
LIN {X 0,Y 323.006,Z 248.248,A -85,B 0,C 180,E1 -15090.764,E2 -15090.764} C_VEL
LIN {X 0,Y 320.607,Z 248.547,A -85,B 0,C 180,E1 -15092.123,E2 -15092.123} C_VEL
LIN {X 0,Y 319.61,Z 248.673,A -85,B 0,C 180,E1 -15093.175,E2 -15093.175} C_VEL
LIN {X 0,Y 319.546,Z 248.676,A -85,B 0,C 180,E1 -15093.531,E2 -15093.531} C_VEL
LIN {X 0,Y 319.585,Z 248.676,A -85,B 0,C 180,E1 -15097.462,E2 -15097.462} C_VEL
LIN {X 0,Y 319.641,Z 248.67,A -85,B 0,C 180,E1 -15100.988,E2 -15100.988} C_VEL
LIN {X 0,Y 319.714,Z 248.66,A -85,B 0,C 180,E1 -15105.289,E2 -15105.289} C_VEL
LIN {X 0,Y 319.726,Z 248.658,A -85,B 0,C 180,E1 -15108.59,E2 -15108.59} C_VEL
LIN {X 0,Y 319.935,Z 248.632,A -85,B 0,C 180,E1 -15112.426,E2 -15112.426} C_VEL
LIN {X 0,Y 319.74,Z 248.657,A -85,B 0,C 180,E1 -15114.956,E2 -15114.956} C_VEL
LIN {X 0,Y 319.964,Z 248.626,A -85,B 0,C 180,E1 -15117.482,E2 -15117.482} C_VEL
LIN {X 0,Y 320.021,Z 248.62,A -85,B 0,C 180,E1 -15121.258,E2 -15121.258} C_VEL
LIN {X 0,Y 319.743,Z 248.654,A -85,B 0,C 180,E1 -15123.781,E2 -15123.781} C_VEL
LIN {X 0,Y 319.938,Z 248.634,A -85,B 0,C 180,E1 -15126.306,E2 -15126.306} C_VEL
LIN {X 0,Y 319.736,Z 248.658,A -85,B 0,C 180,E1 -15130.128,E2 -15130.128} C_VEL
LIN {X 0,Y 319.734,Z 248.659,A -85,B 0,C 180,E1 -15133.992,E2 -15133.992} C_VEL
LIN {X 0,Y 319.661,Z 248.668,A -85,B 0,C 180,E1 -15137.927,E2 -15137.927} C_VEL
LIN {X 0,Y 319.603,Z 248.672,A -85,B 0,C 180,E1 -15140.6,E2 -15140.6} C_VEL
LIN {X 0,Y 319.542,Z 248.681,A -85,B 0,C 180,E1 -15143.322,E2 -15143.322} C_VEL
LIN {X 0,Y 319.553,Z 248.682,A -85,B 0,C 180,E1 -15146.095,E2 -15146.095} C_VEL
LIN {X 0,Y 319.544,Z 248.681,A -85,B 0,C 180,E1 -15148.938,E2 -15148.938} C_VEL
LIN {X 0,Y 319.525,Z 248.686,A -85,B 0,C 180,E1 -15151.863,E2 -15151.863} C_VEL
LIN {X 0,Y 319.581,Z 248.679,A -85,B 0,C 180,E1 -15155.543,E2 -15155.543} C_VEL
LIN {X 0,Y 319.528,Z 248.682,A -85,B 0,C 180,E1 -15159.662,E2 -15159.662} C_VEL
LIN {X 0,Y 319.532,Z 248.771,A -85,B 0,C 180,E1 -15160.869,E2 -15160.869} C_VEL
LIN {X 0,Y 320.474,Z 253.551,A -85,B 0,C 180,E1 -15164.569,E2 -15164.569} C_VEL
LIN {X 0,Y 321.358,Z 258.389,A -85,B 0,C 180,E1 -15168.036,E2 -15168.036} C_VEL
LIN {X 0,Y 322.279,Z 263.904,A -85,B 0,C 180,E1 -15171.726,E2 -15171.726} C_VEL
LIN {X 0,Y 322.366,Z 267.466,A -85,B 0,C 180,E1 -15173.94,E2 -15173.94} C_VEL
LIN {X 0,Y 321.649,Z 272.504,A -85,B 0,C 180,E1 -15176.89,E2 -15176.89} C_VEL
LIN {X 0,Y 320.614,Z 279.973,A -85,B 0,C 180,E1 -15181.168,E2 -15181.168} C_VEL
LIN {X 0,Y 319.708,Z 287.323,A -85,B 0,C 180,E1 -15185.313,E2 -15185.313} C_VEL
LIN {X 0,Y 319.37,Z 290.637,A -85,B 0,C 180,E1 -15187.143,E2 -15187.143} C_VEL
LIN {X 0,Y 322.044,Z 304.03,A -85,B 0,C 180,E1 -15187.87,E2 -15187.87} C_VEL
LIN {X 0,Y 323.814,Z 316.497,A -85,B 0,C 180,E1 -15188.752,E2 -15188.752} C_VEL
LIN {X 0,Y 324.898,Z 327.91,A -85,B 0,C 180,E1 -15189.751,E2 -15189.751} C_VEL
LIN {X 0,Y 325.3,Z 336.17,A -85,B 0,C 180,E1 -15190.599,E2 -15190.599} C_VEL
LIN {X 0,Y 323.707,Z 347.995,A -85,B 0,C 180,E1 -15191.978,E2 -15191.978} C_VEL
LIN {X 0,Y 322.253,Z 358.511,A -85,B 0,C 180,E1 -15193.53,E2 -15193.53} C_VEL
LIN {X 0,Y 321.138,Z 367.039,A -85,B 0,C 180,E1 -15195.099,E2 -15195.099} C_VEL
LIN {X 0,Y 320.001,Z 375.366,A -85,B 0,C 180,E1 -15196.99,E2 -15196.99} C_VEL
LIN {X 0,Y 319.07,Z 382.083,A -85,B 0,C 180,E1 -15198.888,E2 -15198.888} C_VEL
LIN {X 0,Y 318.388,Z 388.244,A -85,B 0,C 180,E1 -15201.111,E2 -15201.111} C_VEL
LIN {X 0,Y 318.093,Z 392.257,A -85,B 0,C 180,E1 -15203.02,E2 -15203.02} C_VEL
LIN {X 0,Y 317.933,Z 395.225,A -85,B 0,C 180,E1 -15204.927,E2 -15204.927} C_VEL
LIN {X 0,Y 317.915,Z 396.642,A -85,B 0,C 180,E1 -15206.198,E2 -15206.198} C_VEL
LIN {X 0,Y 317.946,Z 398.272,A -85,B 0,C 180,E1 -15208.734,E2 -15208.734} C_VEL
LIN {X 0,Y 318.048,Z 398.496,A -85,B 0,C 180,E1 -15210,E2 -15210} C_VEL
LIN {X 0,Y 317.946,Z 398.268,A -85,B 0,C 180,E1 -15211.267,E2 -15211.267} C_VEL
LIN {X 0,Y 317.915,Z 396.636,A -85,B 0,C 180,E1 -15213.803,E2 -15213.803} C_VEL
LIN {X 0,Y 318.001,Z 393.9,A -85,B 0,C 180,E1 -15215.996,E2 -15215.996} C_VEL
LIN {X 0,Y 318.241,Z 389.665,A -85,B 0,C 180,E1 -15218.253,E2 -15218.253} C_VEL
LIN {X 0,Y 318.758,Z 384.895,A -85,B 0,C 180,E1 -15220.159,E2 -15220.159} C_VEL
LIN {X 0,Y 319.602,Z 377.737,A -85,B 0,C 180,E1 -15222.381,E2 -15222.381} C_VEL
LIN {X 0,Y 320.734,Z 369.985,A -85,B 0,C 180,E1 -15224.272,E2 -15224.272} C_VEL
LIN {X 0,Y 322.03,Z 360.914,A -85,B 0,C 180,E1 -15226.038,E2 -15226.038} C_VEL
LIN {X 0,Y 323.198,Z 351.307,A -85,B 0,C 180,E1 -15227.561,E2 -15227.561} C_VEL
LIN {X 0,Y 324.75,Z 340.359,A -85,B 0,C 180,E1 -15228.943,E2 -15228.943} C_VEL
LIN {X 0,Y 325.344,Z 334.506,A -85,B 0,C 180,E1 -15229.562,E2 -15229.562} C_VEL
LIN {X 0,Y 324.404,Z 322.414,A -85,B 0,C 180,E1 -15230.744,E2 -15230.744} C_VEL
LIN {X 0,Y 322.985,Z 310.137,A -85,B 0,C 180,E1 -15231.711,E2 -15231.711} C_VEL
LIN {X 0,Y 320.777,Z 297.399,A -85,B 0,C 180,E1 -15232.505,E2 -15232.505} C_VEL
LIN {X 0,Y 319.379,Z 290.503,A -85,B 0,C 180,E1 -15232.861,E2 -15232.861} C_VEL
LIN {X 0,Y 320.125,Z 283.647,A -85,B 0,C 180,E1 -15236.748,E2 -15236.748} C_VEL
LIN {X 0,Y 320.927,Z 277.467,A -85,B 0,C 180,E1 -15240.244,E2 -15240.244} C_VEL
LIN {X 0,Y 321.894,Z 271.035,A -85,B 0,C 180,E1 -15243.936,E2 -15243.936} C_VEL
LIN {X 0,Y 322.451,Z 266.063,A -85,B 0,C 180,E1 -15246.856,E2 -15246.856} C_VEL
LIN {X 0,Y 322.023,Z 262.276,A -85,B 0,C 180,E1 -15249.266,E2 -15249.266} C_VEL
LIN {X 0,Y 321.132,Z 257.174,A -85,B 0,C 180,E1 -15252.722,E2 -15252.722} C_VEL
LIN {X 0,Y 320.214,Z 252.167,A -85,B 0,C 180,E1 -15256.41,E2 -15256.41} C_VEL
LIN {X 0,Y 319.533,Z 248.684,A -85,B 0,C 180,E1 -15259.235,E2 -15259.235} C_VEL
LIN {X 0,Y 319.559,Z 248.679,A -85,B 0,C 180,E1 -15263.572,E2 -15263.572} C_VEL
LIN {X 0,Y 319.58,Z 248.679,A -85,B 0,C 180,E1 -15266.687,E2 -15266.687} C_VEL
LIN {X 0,Y 319.563,Z 248.677,A -85,B 0,C 180,E1 -15269.614,E2 -15269.614} C_VEL
LIN {X 0,Y 319.542,Z 248.683,A -85,B 0,C 180,E1 -15272.492,E2 -15272.492} C_VEL
LIN {X 0,Y 319.544,Z 248.68,A -85,B 0,C 180,E1 -15275.299,E2 -15275.299} C_VEL
LIN {X 0,Y 319.568,Z 248.681,A -85,B 0,C 180,E1 -15278.046,E2 -15278.046} C_VEL
LIN {X 0,Y 319.692,Z 248.661,A -85,B 0,C 180,E1 -15280.963,E2 -15280.963} C_VEL
LIN {X 0,Y 319.735,Z 248.656,A -85,B 0,C 180,E1 -15285.276,E2 -15285.276} C_VEL
LIN {X 0,Y 319.716,Z 248.658,A -85,B 0,C 180,E1 -15288.589,E2 -15288.589} C_VEL
LIN {X 0,Y 319.898,Z 248.635,A -85,B 0,C 180,E1 -15292.425,E2 -15292.425} C_VEL
LIN {X 0,Y 319.746,Z 248.654,A -85,B 0,C 180,E1 -15294.956,E2 -15294.956} C_VEL
LIN {X 0,Y 319.993,Z 248.628,A -85,B 0,C 180,E1 -15297.482,E2 -15297.482} C_VEL
LIN {X 0,Y 320.003,Z 248.625,A -85,B 0,C 180,E1 -15301.259,E2 -15301.259} C_VEL
LIN {X 0,Y 319.719,Z 248.659,A -85,B 0,C 180,E1 -15303.781,E2 -15303.781} C_VEL
LIN {X 0,Y 319.902,Z 248.632,A -85,B 0,C 180,E1 -15306.617,E2 -15306.617} C_VEL
LIN {X 0,Y 319.74,Z 248.654,A -85,B 0,C 180,E1 -15310.128,E2 -15310.128} C_VEL
LIN {X 0,Y 319.736,Z 248.655,A -85,B 0,C 180,E1 -15313.992,E2 -15313.992} C_VEL
LIN {X 0,Y 319.628,Z 248.667,A -85,B 0,C 180,E1 -15317.929,E2 -15317.929} C_VEL
LIN {X 0,Y 319.571,Z 248.675,A -85,B 0,C 180,E1 -15321.954,E2 -15321.954} C_VEL
LIN {X 0,Y 319.574,Z 248.676,A -85,B 0,C 180,E1 -15326.094,E2 -15326.094} C_VEL
LIN {X 0,Y 319.546,Z 248.681,A -85,B 0,C 180,E1 -15328.938,E2 -15328.938} C_VEL
LIN {X 0,Y 319.527,Z 248.682,A -85,B 0,C 180,E1 -15331.863,E2 -15331.863} C_VEL
LIN {X 0,Y 319.583,Z 248.673,A -85,B 0,C 180,E1 -15335.543,E2 -15335.543} C_VEL
LIN {X 0,Y 319.576,Z 248.678,A -85,B 0,C 180,E1 -15338.008,E2 -15338.008} C_VEL
LIN {X 0,Y 319.529,Z 248.682,A -85,B 0,C 180,E1 -15341.597,E2 -15341.597} C_VEL
LIN {X 0,Y 319.491,Z 248.685,A -85,B 0,C 180,E1 -15345.257,E2 -15345.257} C_VEL
LIN {X 0,Y 319.53,Z 248.681,A -85,B 0,C 180,E1 -15348.711,E2 -15348.711} C_VEL
LIN {X 0,Y 319.538,Z 248.681,A -85,B 0,C 180,E1 -15352.354,E2 -15352.354} C_VEL
LIN {X 0,Y 319.356,Z 248.703,A -85,B 0,C 180,E1 -15355.097,E2 -15355.097} C_VEL
LIN {X 0,Y 319.167,Z 248.73,A -85,B 0,C 180,E1 -15356.799,E2 -15356.799} C_VEL
LIN {X 0,Y 319.079,Z 249.261,A -85,B 0,C 180,E1 -15358.087,E2 -15358.087} C_VEL
LIN {X 0,Y 318.972,Z 251.625,A -85,B 0,C 180,E1 -15361.005,E2 -15361.005} C_VEL
LIN {X 0,Y 318.867,Z 255.282,A -85,B 0,C 180,E1 -15365.243,E2 -15365.243} C_VEL
LIN {X 0,Y 318.795,Z 257.07,A -85,B 0,C 180,E1 -15367.211,E2 -15367.211} C_VEL
LIN {X 0,Y 323.22,Z 271.137,A -85,B 0,C 180,E1 -15368.19,E2 -15368.19} C_VEL
LIN {X 0,Y 326.296,Z 283.365,A -85,B 0,C 180,E1 -15369.233,E2 -15369.233} C_VEL
LIN {X 0,Y 327.525,Z 290.37,A -85,B 0,C 180,E1 -15369.92,E2 -15369.92} C_VEL
LIN {X 0,Y 326.454,Z 301.427,A -85,B 0,C 180,E1 -15370.997,E2 -15370.997} C_VEL
LIN {X 0,Y 325.389,Z 311.316,A -85,B 0,C 180,E1 -15372.206,E2 -15372.206} C_VEL
LIN {X 0,Y 324.106,Z 320.819,A -85,B 0,C 180,E1 -15373.626,E2 -15373.626} C_VEL
LIN {X 0,Y 322.842,Z 329.276,A -85,B 0,C 180,E1 -15375.179,E2 -15375.179} C_VEL
LIN {X 0,Y 321.509,Z 337.49,A -85,B 0,C 180,E1 -15377.052,E2 -15377.052} C_VEL
LIN {X 0,Y 320.61,Z 343.105,A -85,B 0,C 180,E1 -15378.621,E2 -15378.621} C_VEL
LIN {X 0,Y 319.767,Z 348.571,A -85,B 0,C 180,E1 -15380.512,E2 -15380.512} C_VEL
LIN {X 0,Y 319.039,Z 353.623,A -85,B 0,C 180,E1 -15382.802,E2 -15382.802} C_VEL
LIN {X 0,Y 318.509,Z 356.972,A -85,B 0,C 180,E1 -15384.936,E2 -15384.936} C_VEL
LIN {X 0,Y 318.406,Z 358.353,A -85,B 0,C 180,E1 -15386.203,E2 -15386.203} C_VEL
LIN {X 0,Y 318.185,Z 359.947,A -85,B 0,C 180,E1 -15388.734,E2 -15388.734} C_VEL
LIN {X 0,Y 318.16,Z 360.177,A -85,B 0,C 180,E1 -15390,E2 -15390} C_VEL
LIN {X 0,Y 318.185,Z 359.987,A -85,B 0,C 180,E1 -15391.265,E2 -15391.265} C_VEL
LIN {X 0,Y 318.285,Z 359.404,A -85,B 0,C 180,E1 -15392.531,E2 -15392.531} C_VEL
LIN {X 0,Y 318.387,Z 358.446,A -85,B 0,C 180,E1 -15393.797,E2 -15393.797} C_VEL
LIN {X 0,Y 318.499,Z 357.103,A -85,B 0,C 180,E1 -15395.064,E2 -15395.064} C_VEL
LIN {X 0,Y 318.961,Z 354.041,A -85,B 0,C 180,E1 -15397.086,E2 -15397.086} C_VEL
LIN {X 0,Y 319.48,Z 350.393,A -85,B 0,C 180,E1 -15398.858,E2 -15398.858} C_VEL
LIN {X 0,Y 320.229,Z 345.408,A -85,B 0,C 180,E1 -15400.751,E2 -15400.751} C_VEL
LIN {X 0,Y 321.277,Z 339.121,A -85,B 0,C 180,E1 -15402.636,E2 -15402.636} C_VEL
LIN {X 0,Y 322.541,Z 331.247,A -85,B 0,C 180,E1 -15404.512,E2 -15404.512} C_VEL
LIN {X 0,Y 323.738,Z 323.218,A -85,B 0,C 180,E1 -15406.069,E2 -15406.069} C_VEL
LIN {X 0,Y 325.12,Z 313.412,A -85,B 0,C 180,E1 -15407.616,E2 -15407.616} C_VEL
LIN {X 0,Y 326.201,Z 303.763,A -85,B 0,C 180,E1 -15408.855,E2 -15408.855} C_VEL
LIN {X 0,Y 327.389,Z 293.297,A -85,B 0,C 180,E1 -15409.925,E2 -15409.925} C_VEL
LIN {X 0,Y 327.608,Z 289.967,A -85,B 0,C 180,E1 -15410.222,E2 -15410.222} C_VEL
LIN {X 0,Y 325.274,Z 278.847,A -85,B 0,C 180,E1 -15411.286,E2 -15411.286} C_VEL
LIN {X 0,Y 321.947,Z 266.703,A -85,B 0,C 180,E1 -15412.253,E2 -15412.253} C_VEL
LIN {X 0,Y 318.799,Z 257.012,A -85,B 0,C 180,E1 -15412.938,E2 -15412.938} C_VEL
LIN {X 0,Y 318.878,Z 254.14,A -85,B 0,C 180,E1 -15416.155,E2 -15416.155} C_VEL
LIN {X 0,Y 318.97,Z 251.734,A -85,B 0,C 180,E1 -15418.995,E2 -15418.995} C_VEL
LIN {X 0,Y 319.077,Z 249.358,A -85,B 0,C 180,E1 -15421.913,E2 -15421.913} C_VEL
LIN {X 0,Y 319.184,Z 248.73,A -85,B 0,C 180,E1 -15423.399,E2 -15423.399} C_VEL
LIN {X 0,Y 319.492,Z 248.691,A -85,B 0,C 180,E1 -15426.437,E2 -15426.437} C_VEL
LIN {X 0,Y 319.56,Z 248.68,A -85,B 0,C 180,E1 -15429.669,E2 -15429.669} C_VEL
LIN {X 0,Y 319.523,Z 248.682,A -85,B 0,C 180,E1 -15433.461,E2 -15433.461} C_VEL
LIN {X 0,Y 319.556,Z 248.676,A -85,B 0,C 180,E1 -15437.016,E2 -15437.016} C_VEL
LIN {X 0,Y 319.548,Z 248.679,A -85,B 0,C 180,E1 -15440.371,E2 -15440.371} C_VEL
LIN {X 0,Y 319.56,Z 248.681,A -85,B 0,C 180,E1 -15443.572,E2 -15443.572} C_VEL
LIN {X 0,Y 319.579,Z 248.674,A -85,B 0,C 180,E1 -15446.686,E2 -15446.686} C_VEL
LIN {X 0,Y 319.562,Z 248.681,A -85,B 0,C 180,E1 -15449.613,E2 -15449.613} C_VEL
LIN {X 0,Y 319.546,Z 248.678,A -85,B 0,C 180,E1 -15452.492,E2 -15452.492} C_VEL
LIN {X 0,Y 319.546,Z 248.676,A -85,B 0,C 180,E1 -15453.531,E2 -15453.531} C_VEL
LIN {X 0,Y 318.925,Z 248.759,A -85,B 0,C 180,E1 -15454.584,E2 -15454.584} C_VEL
LIN {X 0,Y 316.096,Z 249.116,A -85,B 0,C 180,E1 -15456.297,E2 -15456.297} C_VEL
LIN {X 0,Y 313.665,Z 249.417,A -85,B 0,C 180,E1 -15457.686,E2 -15457.686} C_VEL
LIN {X 0,Y 312.612,Z 249.544,A -85,B 0,C 180,E1 -15458.761,E2 -15458.761} C_VEL
LIN {X 0,Y 312.523,Z 249.553,A -85,B 0,C 180,E1 -15459.126,E2 -15459.126} C_VEL
LIN {X 0,Y 312.584,Z 249.546,A -85,B 0,C 180,E1 -15461.653,E2 -15461.653} C_VEL
LIN {X 0,Y 312.687,Z 249.533,A -85,B 0,C 180,E1 -15465.686,E2 -15465.686} C_VEL
LIN {X 0,Y 312.705,Z 249.531,A -85,B 0,C 180,E1 -15469.642,E2 -15469.642} C_VEL
LIN {X 0,Y 312.874,Z 249.51,A -85,B 0,C 180,E1 -15472.254,E2 -15472.254} C_VEL
LIN {X 0,Y 312.711,Z 249.534,A -85,B 0,C 180,E1 -15474.842,E2 -15474.842} C_VEL
LIN {X 0,Y 312.97,Z 249.501,A -85,B 0,C 180,E1 -15478.713,E2 -15478.713} C_VEL
LIN {X 0,Y 312.938,Z 249.505,A -85,B 0,C 180,E1 -15482.574,E2 -15482.574} C_VEL
LIN {X 0,Y 312.894,Z 249.511,A -85,B 0,C 180,E1 -15486.448,E2 -15486.448} C_VEL
LIN {X 0,Y 312.686,Z 249.538,A -85,B 0,C 180,E1 -15490.359,E2 -15490.359} C_VEL
LIN {X 0,Y 312.702,Z 249.53,A -85,B 0,C 180,E1 -15494.888,E2 -15494.888} C_VEL
LIN {X 0,Y 312.631,Z 249.541,A -85,B 0,C 180,E1 -15499.236,E2 -15499.236} C_VEL
LIN {X 0,Y 312.518,Z 249.555,A -85,B 0,C 180,E1 -15502.776,E2 -15502.776} C_VEL
LIN {X 0,Y 312.487,Z 249.56,A -85,B 0,C 180,E1 -15506.732,E2 -15506.732} C_VEL
LIN {X 0,Y 312.497,Z 249.564,A -85,B 0,C 180,E1 -15509.655,E2 -15509.655} C_VEL
LIN {X 0,Y 312.521,Z 249.559,A -85,B 0,C 180,E1 -15513.689,E2 -15513.689} C_VEL
LIN {X 0,Y 312.515,Z 249.558,A -85,B 0,C 180,E1 -15517.387,E2 -15517.387} C_VEL
LIN {X 0,Y 312.527,Z 249.704,A -85,B 0,C 180,E1 -15520.355,E2 -15520.355} C_VEL
LIN {X 0,Y 313.424,Z 254.442,A -85,B 0,C 180,E1 -15524.148,E2 -15524.148} C_VEL
LIN {X 0,Y 314.337,Z 259.501,A -85,B 0,C 180,E1 -15527.875,E2 -15527.875} C_VEL
LIN {X 0,Y 315.209,Z 264.59,A -85,B 0,C 180,E1 -15531.369,E2 -15531.369} C_VEL
LIN {X 0,Y 315.339,Z 268.63,A -85,B 0,C 180,E1 -15533.961,E2 -15533.961} C_VEL
LIN {X 0,Y 314.625,Z 273.387,A -85,B 0,C 180,E1 -15536.82,E2 -15536.82} C_VEL
LIN {X 0,Y 313.611,Z 280.361,A -85,B 0,C 180,E1 -15540.926,E2 -15540.926} C_VEL
LIN {X 0,Y 312.612,Z 288.115,A -85,B 0,C 180,E1 -15545.423,E2 -15545.423} C_VEL
LIN {X 0,Y 312.38,Z 290.141,A -85,B 0,C 180,E1 -15546.595,E2 -15546.595} C_VEL
LIN {X 0,Y 315.116,Z 303.756,A -85,B 0,C 180,E1 -15547.366,E2 -15547.366} C_VEL
LIN {X 0,Y 316.927,Z 315.878,A -85,B 0,C 180,E1 -15548.253,E2 -15548.253} C_VEL
LIN {X 0,Y 318.003,Z 327.472,A -85,B 0,C 180,E1 -15549.292,E2 -15549.292} C_VEL
LIN {X 0,Y 318.397,Z 337.177,A -85,B 0,C 180,E1 -15550.329,E2 -15550.329} C_VEL
LIN {X 0,Y 316.762,Z 348.749,A -85,B 0,C 180,E1 -15551.736,E2 -15551.736} C_VEL
LIN {X 0,Y 315.404,Z 358.083,A -85,B 0,C 180,E1 -15553.162,E2 -15553.162} C_VEL
LIN {X 0,Y 314.262,Z 366.612,A -85,B 0,C 180,E1 -15554.766,E2 -15554.766} C_VEL
LIN {X 0,Y 313.028,Z 374.937,A -85,B 0,C 180,E1 -15556.695,E2 -15556.695} C_VEL
LIN {X 0,Y 312.049,Z 381.654,A -85,B 0,C 180,E1 -15558.635,E2 -15558.635} C_VEL
LIN {X 0,Y 311.361,Z 387.816,A -85,B 0,C 180,E1 -15560.909,E2 -15560.909} C_VEL
LIN {X 0,Y 311.021,Z 391.829,A -85,B 0,C 180,E1 -15562.861,E2 -15562.861} C_VEL
LIN {X 0,Y 310.85,Z 394.798,A -85,B 0,C 180,E1 -15564.811,E2 -15564.811} C_VEL
LIN {X 0,Y 310.845,Z 396.215,A -85,B 0,C 180,E1 -15566.111,E2 -15566.111} C_VEL
LIN {X 0,Y 310.853,Z 397.845,A -85,B 0,C 180,E1 -15568.705,E2 -15568.705} C_VEL
LIN {X 0,Y 310.959,Z 398.069,A -85,B 0,C 180,E1 -15570,E2 -15570} C_VEL
LIN {X 0,Y 310.853,Z 397.841,A -85,B 0,C 180,E1 -15571.296,E2 -15571.296} C_VEL
LIN {X 0,Y 310.845,Z 396.209,A -85,B 0,C 180,E1 -15573.889,E2 -15573.889} C_VEL
LIN {X 0,Y 310.899,Z 393.748,A -85,B 0,C 180,E1 -15575.935,E2 -15575.935} C_VEL
LIN {X 0,Y 311.064,Z 390.565,A -85,B 0,C 180,E1 -15577.791,E2 -15577.791} C_VEL
LIN {X 0,Y 311.522,Z 386.178,A -85,B 0,C 180,E1 -15579.742,E2 -15579.742} C_VEL
LIN {X 0,Y 312.157,Z 380.594,A -85,B 0,C 180,E1 -15581.691,E2 -15581.691} C_VEL
LIN {X 0,Y 313.229,Z 373.647,A -85,B 0,C 180,E1 -15583.627,E2 -15583.627} C_VEL
LIN {X 0,Y 314.285,Z 366.556,A -85,B 0,C 180,E1 -15585.234,E2 -15585.234} C_VEL
LIN {X 0,Y 315.46,Z 358.014,A -85,B 0,C 180,E1 -15586.836,E2 -15586.836} C_VEL
LIN {X 0,Y 316.938,Z 347.475,A -85,B 0,C 180,E1 -15588.421,E2 -15588.421} C_VEL
LIN {X 0,Y 318.418,Z 337.066,A -85,B 0,C 180,E1 -15589.67,E2 -15589.67} C_VEL
LIN {X 0,Y 317.878,Z 325.821,A -85,B 0,C 180,E1 -15590.859,E2 -15590.859} C_VEL
LIN {X 0,Y 316.493,Z 312.821,A -85,B 0,C 180,E1 -15591.976,E2 -15591.976} C_VEL
LIN {X 0,Y 314.39,Z 299.767,A -85,B 0,C 180,E1 -15592.863,E2 -15592.863} C_VEL
LIN {X 0,Y 312.354,Z 290.072,A -85,B 0,C 180,E1 -15593.392,E2 -15593.392} C_VEL
LIN {X 0,Y 313.193,Z 283.24,A -85,B 0,C 180,E1 -15597.389,E2 -15597.389} C_VEL
LIN {X 0,Y 314.027,Z 277.082,A -85,B 0,C 180,E1 -15600.981,E2 -15600.981} C_VEL
LIN {X 0,Y 314.932,Z 271.412,A -85,B 0,C 180,E1 -15604.341,E2 -15604.341} C_VEL
LIN {X 0,Y 315.455,Z 267.051,A -85,B 0,C 180,E1 -15606.98,E2 -15606.98} C_VEL
LIN {X 0,Y 314.994,Z 263.21,A -85,B 0,C 180,E1 -15609.485,E2 -15609.485} C_VEL
LIN {X 0,Y 314.036,Z 257.781,A -85,B 0,C 180,E1 -15613.275,E2 -15613.275} C_VEL
LIN {X 0,Y 313.158,Z 253.119,A -85,B 0,C 180,E1 -15616.804,E2 -15616.804} C_VEL
LIN {X 0,Y 312.503,Z 249.557,A -85,B 0,C 180,E1 -15619.876,E2 -15619.876} C_VEL
LIN {X 0,Y 312.537,Z 249.555,A -85,B 0,C 180,E1 -15624.051,E2 -15624.051} C_VEL
LIN {X 0,Y 312.504,Z 249.557,A -85,B 0,C 180,E1 -15627.334,E2 -15627.334} C_VEL
LIN {X 0,Y 312.509,Z 249.555,A -85,B 0,C 180,E1 -15631.292,E2 -15631.292} C_VEL
LIN {X 0,Y 312.525,Z 249.556,A -85,B 0,C 180,E1 -15634.706,E2 -15634.706} C_VEL
LIN {X 0,Y 312.538,Z 249.553,A -85,B 0,C 180,E1 -15638.913,E2 -15638.913} C_VEL
LIN {X 0,Y 312.642,Z 249.542,A -85,B 0,C 180,E1 -15641.657,E2 -15641.657} C_VEL
LIN {X 0,Y 312.697,Z 249.535,A -85,B 0,C 180,E1 -15645.686,E2 -15645.686} C_VEL
LIN {X 0,Y 312.688,Z 249.537,A -85,B 0,C 180,E1 -15649.641,E2 -15649.641} C_VEL
LIN {X 0,Y 312.896,Z 249.511,A -85,B 0,C 180,E1 -15653.552,E2 -15653.552} C_VEL
LIN {X 0,Y 312.94,Z 249.506,A -85,B 0,C 180,E1 -15657.426,E2 -15657.426} C_VEL
LIN {X 0,Y 312.972,Z 249.501,A -85,B 0,C 180,E1 -15661.287,E2 -15661.287} C_VEL
LIN {X 0,Y 312.706,Z 249.535,A -85,B 0,C 180,E1 -15665.158,E2 -15665.158} C_VEL
LIN {X 0,Y 312.834,Z 249.516,A -85,B 0,C 180,E1 -15667.747,E2 -15667.747} C_VEL
LIN {X 0,Y 312.668,Z 249.535,A -85,B 0,C 180,E1 -15671.671,E2 -15671.671} C_VEL
LIN {X 0,Y 312.671,Z 249.539,A -85,B 0,C 180,E1 -15674.865,E2 -15674.865} C_VEL
LIN {X 0,Y 312.589,Z 249.547,A -85,B 0,C 180,E1 -15679.213,E2 -15679.213} C_VEL
LIN {X 0,Y 312.526,Z 249.557,A -85,B 0,C 180,E1 -15682.779,E2 -15682.779} C_VEL
LIN {X 0,Y 312.534,Z 249.552,A -85,B 0,C 180,E1 -15685.908,E2 -15685.908} C_VEL
LIN {X 0,Y 312.499,Z 249.556,A -85,B 0,C 180,E1 -15689.655,E2 -15689.655} C_VEL
LIN {X 0,Y 312.523,Z 249.554,A -85,B 0,C 180,E1 -15693.689,E2 -15693.689} C_VEL
LIN {X 0,Y 312.529,Z 249.553,A -85,B 0,C 180,E1 -15697.385,E2 -15697.385} C_VEL
LIN {X 0,Y 312.493,Z 249.559,A -85,B 0,C 180,E1 -15700.709,E2 -15700.709} C_VEL
LIN {X 0,Y 312.455,Z 249.566,A -85,B 0,C 180,E1 -15704.209,E2 -15704.209} C_VEL
LIN {X 0,Y 312.486,Z 249.562,A -85,B 0,C 180,E1 -15707.919,E2 -15707.919} C_VEL
LIN {X 0,Y 312.478,Z 249.559,A -85,B 0,C 180,E1 -15710.968,E2 -15710.968} C_VEL
LIN {X 0,Y 312.403,Z 249.57,A -85,B 0,C 180,E1 -15714.203,E2 -15714.203} C_VEL
LIN {X 0,Y 312.052,Z 249.657,A -85,B 0,C 180,E1 -15717.28,E2 -15717.28} C_VEL
LIN {X 0,Y 311.965,Z 252.032,A -85,B 0,C 180,E1 -15720.289,E2 -15720.289} C_VEL
LIN {X 0,Y 311.861,Z 254.458,A -85,B 0,C 180,E1 -15723.21,E2 -15723.21} C_VEL
LIN {X 0,Y 311.758,Z 257.516,A -85,B 0,C 180,E1 -15726.652,E2 -15726.652} C_VEL
LIN {X 0,Y 316.506,Z 272.346,A -85,B 0,C 180,E1 -15727.746,E2 -15727.746} C_VEL
LIN {X 0,Y 319.514,Z 284.352,A -85,B 0,C 180,E1 -15728.815,E2 -15728.815} C_VEL
LIN {X 0,Y 320.813,Z 290.808,A -85,B 0,C 180,E1 -15729.481,E2 -15729.481} C_VEL
LIN {X 0,Y 319.782,Z 301.858,A -85,B 0,C 180,E1 -15730.585,E2 -15730.585} C_VEL
LIN {X 0,Y 318.627,Z 311.922,A -85,B 0,C 180,E1 -15731.84,E2 -15731.84} C_VEL
LIN {X 0,Y 317.311,Z 321.25,A -85,B 0,C 180,E1 -15733.266,E2 -15733.266} C_VEL
LIN {X 0,Y 315.995,Z 329.706,A -85,B 0,C 180,E1 -15734.851,E2 -15734.851} C_VEL
LIN {X 0,Y 314.623,Z 337.918,A -85,B 0,C 180,E1 -15736.764,E2 -15736.764} C_VEL
LIN {X 0,Y 313.681,Z 343.532,A -85,B 0,C 180,E1 -15738.367,E2 -15738.367} C_VEL
LIN {X 0,Y 312.761,Z 349,A -85,B 0,C 180,E1 -15740.297,E2 -15740.297} C_VEL
LIN {X 0,Y 312.096,Z 353.287,A -85,B 0,C 180,E1 -15742.235,E2 -15742.235} C_VEL
LIN {X 0,Y 311.79,Z 355.552,A -85,B 0,C 180,E1 -15743.529,E2 -15743.529} C_VEL
LIN {X 0,Y 311.459,Z 357.399,A -85,B 0,C 180,E1 -15744.821,E2 -15744.821} C_VEL
LIN {X 0,Y 311.327,Z 358.781,A -85,B 0,C 180,E1 -15746.117,E2 -15746.117} C_VEL
LIN {X 0,Y 311.115,Z 360.373,A -85,B 0,C 180,E1 -15748.705,E2 -15748.705} C_VEL
LIN {X 0,Y 311.086,Z 360.603,A -85,B 0,C 180,E1 -15750,E2 -15750} C_VEL
LIN {X 0,Y 311.114,Z 360.412,A -85,B 0,C 180,E1 -15751.294,E2 -15751.294} C_VEL
LIN {X 0,Y 311.308,Z 358.872,A -85,B 0,C 180,E1 -15753.883,E2 -15753.883} C_VEL
LIN {X 0,Y 311.448,Z 357.529,A -85,B 0,C 180,E1 -15755.179,E2 -15755.179} C_VEL
LIN {X 0,Y 311.897,Z 354.69,A -85,B 0,C 180,E1 -15757.113,E2 -15757.113} C_VEL
LIN {X 0,Y 312.488,Z 350.818,A -85,B 0,C 180,E1 -15759.058,E2 -15759.058} C_VEL
LIN {X 0,Y 313.273,Z 345.833,A -85,B 0,C 180,E1 -15760.993,E2 -15760.993} C_VEL
LIN {X 0,Y 314.375,Z 339.545,A -85,B 0,C 180,E1 -15762.918,E2 -15762.918} C_VEL
LIN {X 0,Y 315.688,Z 331.671,A -85,B 0,C 180,E1 -15764.834,E2 -15764.834} C_VEL
LIN {X 0,Y 316.952,Z 323.641,A -85,B 0,C 180,E1 -15766.422,E2 -15766.422} C_VEL
LIN {X 0,Y 318.389,Z 313.834,A -85,B 0,C 180,E1 -15768.001,E2 -15768.001} C_VEL
LIN {X 0,Y 319.527,Z 304.184,A -85,B 0,C 180,E1 -15769.264,E2 -15769.264} C_VEL
LIN {X 0,Y 320.742,Z 293.717,A -85,B 0,C 180,E1 -15770.356,E2 -15770.356} C_VEL
LIN {X 0,Y 320.774,Z 290.541,A -85,B 0,C 180,E1 -15770.658,E2 -15770.658} C_VEL
LIN {X 0,Y 318.342,Z 279.186,A -85,B 0,C 180,E1 -15771.78,E2 -15771.78} C_VEL
LIN {X 0,Y 314.921,Z 266.999,A -85,B 0,C 180,E1 -15772.784,E2 -15772.784} C_VEL
LIN {X 0,Y 311.745,Z 257.458,A -85,B 0,C 180,E1 -15773.476,E2 -15773.476} C_VEL
LIN {X 0,Y 311.851,Z 254.559,A -85,B 0,C 180,E1 -15776.79,E2 -15776.79} C_VEL
LIN {X 0,Y 311.964,Z 252.142,A -85,B 0,C 180,E1 -15779.711,E2 -15779.711} C_VEL
LIN {X 0,Y 312.056,Z 249.757,A -85,B 0,C 180,E1 -15782.719,E2 -15782.719} C_VEL
LIN {X 0,Y 312.427,Z 249.569,A -85,B 0,C 180,E1 -15785.922,E2 -15785.922} C_VEL
LIN {X 0,Y 312.477,Z 249.561,A -85,B 0,C 180,E1 -15789.032,E2 -15789.032} C_VEL
LIN {X 0,Y 312.491,Z 249.56,A -85,B 0,C 180,E1 -15792.431,E2 -15792.431} C_VEL
LIN {X 0,Y 312.46,Z 249.564,A -85,B 0,C 180,E1 -15796.035,E2 -15796.035} C_VEL
LIN {X 0,Y 312.505,Z 249.56,A -85,B 0,C 180,E1 -15799.875,E2 -15799.875} C_VEL
LIN {X 0,Y 312.527,Z 249.553,A -85,B 0,C 180,E1 -15802.615,E2 -15802.615} C_VEL
LIN {X 0,Y 312.521,Z 249.554,A -85,B 0,C 180,E1 -15806.311,E2 -15806.311} C_VEL
LIN {X 0,Y 312.498,Z 249.557,A -85,B 0,C 180,E1 -15810.345,E2 -15810.345} C_VEL
LIN {X 0,Y 312.531,Z 249.552,A -85,B 0,C 180,E1 -15814.092,E2 -15814.092} C_VEL
LIN {X 0,Y 312.565,Z 249.55,A -85,B 0,C 180,E1 -15817.527,E2 -15817.527} C_VEL
LIN {X 0,Y 312.523,Z 249.553,A -85,B 0,C 180,E1 -15819.126,E2 -15819.126} C_VEL
LIN {X 0,Y 311.842,Z 249.639,A -85,B 0,C 180,E1 -15820.202,E2 -15820.202} C_VEL
LIN {X 0,Y 308.986,Z 249.993,A -85,B 0,C 180,E1 -15821.954,E2 -15821.954} C_VEL
LIN {X 0,Y 306.611,Z 250.293,A -85,B 0,C 180,E1 -15823.375,E2 -15823.375} C_VEL
LIN {X 0,Y 305.647,Z 250.411,A -85,B 0,C 180,E1 -15824.476,E2 -15824.476} C_VEL
LIN {X 0,Y 305.597,Z 250.418,A -85,B 0,C 180,E1 -15824.848,E2 -15824.848} C_VEL
LIN {X 0,Y 305.606,Z 250.415,A -85,B 0,C 180,E1 -15828.055,E2 -15828.055} C_VEL
LIN {X 0,Y 305.815,Z 250.389,A -85,B 0,C 180,E1 -15832.074,E2 -15832.074} C_VEL
LIN {X 0,Y 305.684,Z 250.41,A -85,B 0,C 180,E1 -15834.723,E2 -15834.723} C_VEL
LIN {X 0,Y 305.938,Z 250.377,A -85,B 0,C 180,E1 -15838.684,E2 -15838.684} C_VEL
LIN {X 0,Y 305.956,Z 250.372,A -85,B 0,C 180,E1 -15841.316,E2 -15841.316} C_VEL
LIN {X 0,Y 305.686,Z 250.405,A -85,B 0,C 180,E1 -15845.277,E2 -15845.277} C_VEL
LIN {X 0,Y 305.774,Z 250.396,A -85,B 0,C 180,E1 -15847.927,E2 -15847.927} C_VEL
LIN {X 0,Y 305.599,Z 250.419,A -85,B 0,C 180,E1 -15851.945,E2 -15851.945} C_VEL
LIN {X 0,Y 305.64,Z 250.41,A -85,B 0,C 180,E1 -15855.035,E2 -15855.035} C_VEL
LIN {X 0,Y 305.577,Z 250.42,A -85,B 0,C 180,E1 -15859.444,E2 -15859.444} C_VEL
LIN {X 0,Y 305.456,Z 250.435,A -85,B 0,C 180,E1 -15863.025,E2 -15863.025} C_VEL
LIN {X 0,Y 305.454,Z 250.438,A -85,B 0,C 180,E1 -15866.191,E2 -15866.191} C_VEL
LIN {X 0,Y 305.45,Z 250.438,A -85,B 0,C 180,E1 -15869.034,E2 -15869.034} C_VEL
LIN {X 0,Y 305.438,Z 250.441,A -85,B 0,C 180,E1 -15871.953,E2 -15871.953} C_VEL
LIN {X 0,Y 305.463,Z 250.437,A -85,B 0,C 180,E1 -15875.113,E2 -15875.113} C_VEL
LIN {X 0,Y 305.46,Z 250.433,A -85,B 0,C 180,E1 -15879.467,E2 -15879.467} C_VEL
LIN {X 0,Y 305.65,Z 251.603,A -85,B 0,C 180,E1 -15880.642,E2 -15880.642} C_VEL
LIN {X 0,Y 306.617,Z 256.634,A -85,B 0,C 180,E1 -15884.72,E2 -15884.72} C_VEL
LIN {X 0,Y 307.668,Z 262.277,A -85,B 0,C 180,E1 -15888.922,E2 -15888.922} C_VEL
LIN {X 0,Y 308.328,Z 266.745,A -85,B 0,C 180,E1 -15892.016,E2 -15892.016} C_VEL
LIN {X 0,Y 308.218,Z 270.529,A -85,B 0,C 180,E1 -15894.447,E2 -15894.447} C_VEL
LIN {X 0,Y 307.318,Z 275.978,A -85,B 0,C 180,E1 -15897.795,E2 -15897.795} C_VEL
LIN {X 0,Y 306.278,Z 282.862,A -85,B 0,C 180,E1 -15901.94,E2 -15901.94} C_VEL
LIN {X 0,Y 305.381,Z 289.692,A -85,B 0,C 180,E1 -15906.015,E2 -15906.015} C_VEL
LIN {X 0,Y 308.314,Z 303.903,A -85,B 0,C 180,E1 -15906.871,E2 -15906.871} C_VEL
LIN {X 0,Y 310.111,Z 315.949,A -85,B 0,C 180,E1 -15907.789,E2 -15907.789} C_VEL
LIN {X 0,Y 311.245,Z 328.827,A -85,B 0,C 180,E1 -15908.994,E2 -15908.994} C_VEL
LIN {X 0,Y 311.667,Z 336.75,A -85,B 0,C 180,E1 -15909.886,E2 -15909.886} C_VEL
LIN {X 0,Y 310.018,Z 348.324,A -85,B 0,C 180,E1 -15911.325,E2 -15911.325} C_VEL
LIN {X 0,Y 308.58,Z 357.656,A -85,B 0,C 180,E1 -15912.778,E2 -15912.778} C_VEL
LIN {X 0,Y 307.396,Z 366.185,A -85,B 0,C 180,E1 -15914.417,E2 -15914.417} C_VEL
LIN {X 0,Y 306.087,Z 374.509,A -85,B 0,C 180,E1 -15916.388,E2 -15916.388} C_VEL
LIN {X 0,Y 305.024,Z 381.223,A -85,B 0,C 180,E1 -15918.369,E2 -15918.369} C_VEL
LIN {X 0,Y 304.308,Z 387.387,A -85,B 0,C 180,E1 -15920.697,E2 -15920.697} C_VEL
LIN {X 0,Y 303.948,Z 391.4,A -85,B 0,C 180,E1 -15922.694,E2 -15922.694} C_VEL
LIN {X 0,Y 303.77,Z 394.37,A -85,B 0,C 180,E1 -15924.69,E2 -15924.69} C_VEL
LIN {X 0,Y 303.754,Z 395.788,A -85,B 0,C 180,E1 -15926.02,E2 -15926.02} C_VEL
LIN {X 0,Y 303.76,Z 397.418,A -85,B 0,C 180,E1 -15928.674,E2 -15928.674} C_VEL
LIN {X 0,Y 303.87,Z 397.642,A -85,B 0,C 180,E1 -15930,E2 -15930} C_VEL
LIN {X 0,Y 303.76,Z 397.414,A -85,B 0,C 180,E1 -15931.326,E2 -15931.326} C_VEL
LIN {X 0,Y 303.754,Z 395.78,A -85,B 0,C 180,E1 -15933.98,E2 -15933.98} C_VEL
LIN {X 0,Y 303.831,Z 393.517,A -85,B 0,C 180,E1 -15935.93,E2 -15935.93} C_VEL
LIN {X 0,Y 304.017,Z 390.135,A -85,B 0,C 180,E1 -15937.973,E2 -15937.973} C_VEL
LIN {X 0,Y 304.481,Z 385.746,A -85,B 0,C 180,E1 -15939.969,E2 -15939.969} C_VEL
LIN {X 0,Y 305.167,Z 380.163,A -85,B 0,C 180,E1 -15941.963,E2 -15941.963} C_VEL
LIN {X 0,Y 306.306,Z 373.215,A -85,B 0,C 180,E1 -15943.941,E2 -15943.941} C_VEL
LIN {X 0,Y 307.418,Z 366.125,A -85,B 0,C 180,E1 -15945.583,E2 -15945.583} C_VEL
LIN {X 0,Y 308.618,Z 357.58,A -85,B 0,C 180,E1 -15947.22,E2 -15947.22} C_VEL
LIN {X 0,Y 309.994,Z 348.221,A -85,B 0,C 180,E1 -15948.677,E2 -15948.677} C_VEL
LIN {X 0,Y 311.636,Z 336.627,A -85,B 0,C 180,E1 -15950.116,E2 -15950.116} C_VEL
LIN {X 0,Y 310.893,Z 324.872,A -85,B 0,C 180,E1 -15951.398,E2 -15951.398} C_VEL
LIN {X 0,Y 309.656,Z 312.646,A -85,B 0,C 180,E1 -15952.468,E2 -15952.468} C_VEL
LIN {X 0,Y 307.441,Z 299.287,A -85,B 0,C 180,E1 -15953.411,E2 -15953.411} C_VEL
LIN {X 0,Y 305.379,Z 289.674,A -85,B 0,C 180,E1 -15953.953,E2 -15953.953} C_VEL
LIN {X 0,Y 306.27,Z 282.831,A -85,B 0,C 180,E1 -15958.062,E2 -15958.062} C_VEL
LIN {X 0,Y 307.314,Z 275.943,A -85,B 0,C 180,E1 -15962.204,E2 -15962.204} C_VEL
LIN {X 0,Y 308.208,Z 270.487,A -85,B 0,C 180,E1 -15965.555,E2 -15965.555} C_VEL
LIN {X 0,Y 308.428,Z 268.006,A -85,B 0,C 180,E1 -15967.105,E2 -15967.105} C_VEL
LIN {X 0,Y 307.962,Z 264.108,A -85,B 0,C 180,E1 -15969.717,E2 -15969.717} C_VEL
LIN {X 0,Y 307.055,Z 259.03,A -85,B 0,C 180,E1 -15973.366,E2 -15973.366} C_VEL
LIN {X 0,Y 306.103,Z 254.032,A -85,B 0,C 180,E1 -15977.283,E2 -15977.283} C_VEL
LIN {X 0,Y 305.458,Z 250.436,A -85,B 0,C 180,E1 -15980.32,E2 -15980.32} C_VEL
LIN {X 0,Y 305.466,Z 250.436,A -85,B 0,C 180,E1 -15983.636,E2 -15983.636} C_VEL
LIN {X 0,Y 305.468,Z 250.438,A -85,B 0,C 180,E1 -15986.483,E2 -15986.483} C_VEL
LIN {X 0,Y 305.433,Z 250.438,A -85,B 0,C 180,E1 -15989.588,E2 -15989.588} C_VEL
LIN {X 0,Y 305.454,Z 250.438,A -85,B 0,C 180,E1 -15992.602,E2 -15992.602} C_VEL
LIN {X 0,Y 305.458,Z 250.436,A -85,B 0,C 180,E1 -15995.534,E2 -15995.534} C_VEL
LIN {X 0,Y 305.509,Z 250.431,A -85,B 0,C 180,E1 -15999.814,E2 -15999.814} C_VEL
LIN {X 0,Y 305.578,Z 250.42,A -85,B 0,C 180,E1 -16002.603,E2 -16002.603} C_VEL
LIN {X 0,Y 305.653,Z 250.411,A -85,B 0,C 180,E1 -16005.349,E2 -16005.349} C_VEL
LIN {X 0,Y 305.627,Z 250.415,A -85,B 0,C 180,E1 -16009.399,E2 -16009.399} C_VEL
LIN {X 0,Y 305.776,Z 250.396,A -85,B 0,C 180,E1 -16012.073,E2 -16012.073} C_VEL
LIN {X 0,Y 305.687,Z 250.405,A -85,B 0,C 180,E1 -16014.723,E2 -16014.723} C_VEL
LIN {X 0,Y 305.958,Z 250.371,A -85,B 0,C 180,E1 -16018.684,E2 -16018.684} C_VEL
LIN {X 0,Y 305.94,Z 250.377,A -85,B 0,C 180,E1 -16021.316,E2 -16021.316} C_VEL
LIN {X 0,Y 305.825,Z 250.387,A -85,B 0,C 180,E1 -16026.598,E2 -16026.598} C_VEL
LIN {X 0,Y 305.698,Z 250.407,A -85,B 0,C 180,E1 -16029.261,E2 -16029.261} C_VEL
LIN {X 0,Y 305.592,Z 250.42,A -85,B 0,C 180,E1 -16033.296,E2 -16033.296} C_VEL
LIN {X 0,Y 305.555,Z 250.421,A -85,B 0,C 180,E1 -16036.022,E2 -16036.022} C_VEL
LIN {X 0,Y 305.546,Z 250.424,A -85,B 0,C 180,E1 -16039.426,E2 -16039.426} C_VEL
LIN {X 0,Y 305.49,Z 250.432,A -85,B 0,C 180,E1 -16043.039,E2 -16043.039} C_VEL
LIN {X 0,Y 305.474,Z 250.433,A -85,B 0,C 180,E1 -16046.197,E2 -16046.197} C_VEL
LIN {X 0,Y 305.452,Z 250.436,A -85,B 0,C 180,E1 -16049.034,E2 -16049.034} C_VEL
LIN {X 0,Y 305.439,Z 250.437,A -85,B 0,C 180,E1 -16051.953,E2 -16051.953} C_VEL
LIN {X 0,Y 305.466,Z 250.432,A -85,B 0,C 180,E1 -16055.113,E2 -16055.113} C_VEL
LIN {X 0,Y 305.47,Z 250.434,A -85,B 0,C 180,E1 -16058.533,E2 -16058.533} C_VEL
LIN {X 0,Y 305.458,Z 250.435,A -85,B 0,C 180,E1 -16062.586,E2 -16062.586} C_VEL
LIN {X 0,Y 305.428,Z 250.439,A -85,B 0,C 180,E1 -16066.345,E2 -16066.345} C_VEL
LIN {X 0,Y 305.46,Z 250.438,A -85,B 0,C 180,E1 -16069.892,E2 -16069.892} C_VEL
LIN {X 0,Y 305.385,Z 250.446,A -85,B 0,C 180,E1 -16073.657,E2 -16073.657} C_VEL
LIN {X 0,Y 305.117,Z 250.479,A -85,B 0,C 180,E1 -16076.44,E2 -16076.44} C_VEL
LIN {X 0,Y 305.025,Z 251.612,A -85,B 0,C 180,E1 -16078.486,E2 -16078.486} C_VEL
LIN {X 0,Y 304.841,Z 254.882,A -85,B 0,C 180,E1 -16082.542,E2 -16082.542} C_VEL
LIN {X 0,Y 304.766,Z 257.971,A -85,B 0,C 180,E1 -16086.103,E2 -16086.103} C_VEL
LIN {X 0,Y 308.979,Z 270.787,A -85,B 0,C 180,E1 -16087.053,E2 -16087.053} C_VEL
LIN {X 0,Y 312.272,Z 283.384,A -85,B 0,C 180,E1 -16088.184,E2 -16088.184} C_VEL
LIN {X 0,Y 313.936,Z 291.258,A -85,B 0,C 180,E1 -16089.011,E2 -16089.011} C_VEL
LIN {X 0,Y 313.964,Z 294.724,A -85,B 0,C 180,E1 -16089.356,E2 -16089.356} C_VEL
LIN {X 0,Y 312.602,Z 306.332,A -85,B 0,C 180,E1 -16090.633,E2 -16090.633} C_VEL
LIN {X 0,Y 311.258,Z 316.742,A -85,B 0,C 180,E1 -16092.082,E2 -16092.082} C_VEL
LIN {X 0,Y 309.929,Z 325.249,A -85,B 0,C 180,E1 -16093.533,E2 -16093.533} C_VEL
LIN {X 0,Y 308.732,Z 333.075,A -85,B 0,C 180,E1 -16095.161,E2 -16095.161} C_VEL
LIN {X 0,Y 307.361,Z 340.727,A -85,B 0,C 180,E1 -16097.118,E2 -16097.118} C_VEL
LIN {X 0,Y 306.047,Z 347.747,A -85,B 0,C 180,E1 -16099.414,E2 -16099.414} C_VEL
LIN {X 0,Y 305.3,Z 352.412,A -85,B 0,C 180,E1 -16101.394,E2 -16101.394} C_VEL
LIN {X 0,Y 304.766,Z 355.979,A -85,B 0,C 180,E1 -16103.379,E2 -16103.379} C_VEL
LIN {X 0,Y 304.412,Z 357.826,A -85,B 0,C 180,E1 -16104.701,E2 -16104.701} C_VEL
LIN {X 0,Y 304.249,Z 359.209,A -85,B 0,C 180,E1 -16106.026,E2 -16106.026} C_VEL
LIN {X 0,Y 304.029,Z 360.8,A -85,B 0,C 180,E1 -16108.675,E2 -16108.675} C_VEL
LIN {X 0,Y 304.014,Z 361.029,A -85,B 0,C 180,E1 -16110,E2 -16110} C_VEL
LIN {X 0,Y 304.029,Z 360.839,A -85,B 0,C 180,E1 -16111.324,E2 -16111.324} C_VEL
LIN {X 0,Y 304.231,Z 359.299,A -85,B 0,C 180,E1 -16113.974,E2 -16113.974} C_VEL
LIN {X 0,Y 304.401,Z 357.955,A -85,B 0,C 180,E1 -16115.299,E2 -16115.299} C_VEL
LIN {X 0,Y 305.031,Z 354.177,A -85,B 0,C 180,E1 -16117.805,E2 -16117.805} C_VEL
LIN {X 0,Y 305.733,Z 349.696,A -85,B 0,C 180,E1 -16119.928,E2 -16119.928} C_VEL
LIN {X 0,Y 306.897,Z 343.291,A -85,B 0,C 180,E1 -16122.229,E2 -16122.229} C_VEL
LIN {X 0,Y 308.11,Z 336.248,A -85,B 0,C 180,E1 -16124.194,E2 -16124.194} C_VEL
LIN {X 0,Y 309.627,Z 327.465,A -85,B 0,C 180,E1 -16126.144,E2 -16126.144} C_VEL
LIN {X 0,Y 311.095,Z 318.444,A -85,B 0,C 180,E1 -16127.757,E2 -16127.757} C_VEL
LIN {X 0,Y 312.418,Z 307.838,A -85,B 0,C 180,E1 -16129.29,E2 -16129.29} C_VEL
LIN {X 0,Y 313.921,Z 295.757,A -85,B 0,C 180,E1 -16130.647,E2 -16130.647} C_VEL
LIN {X 0,Y 314.136,Z 292.391,A -85,B 0,C 180,E1 -16130.975,E2 -16130.975} C_VEL
LIN {X 0,Y 311.927,Z 281.663,A -85,B 0,C 180,E1 -16132.091,E2 -16132.091} C_VEL
LIN {X 0,Y 308.628,Z 269.626,A -85,B 0,C 180,E1 -16133.158,E2 -16133.158} C_VEL
LIN {X 0,Y 304.744,Z 257.902,A -85,B 0,C 180,E1 -16134.039,E2 -16134.039} C_VEL
LIN {X 0,Y 304.833,Z 254.982,A -85,B 0,C 180,E1 -16137.458,E2 -16137.458} C_VEL
LIN {X 0,Y 305.024,Z 251.713,A -85,B 0,C 180,E1 -16141.514,E2 -16141.514} C_VEL
LIN {X 0,Y 305.116,Z 250.481,A -85,B 0,C 180,E1 -16143.56,E2 -16143.56} C_VEL
LIN {X 0,Y 305.391,Z 250.446,A -85,B 0,C 180,E1 -16146.751,E2 -16146.751} C_VEL
LIN {X 0,Y 305.459,Z 250.438,A -85,B 0,C 180,E1 -16150.108,E2 -16150.108} C_VEL
LIN {X 0,Y 305.427,Z 250.44,A -85,B 0,C 180,E1 -16153.655,E2 -16153.655} C_VEL
LIN {X 0,Y 305.456,Z 250.433,A -85,B 0,C 180,E1 -16157.414,E2 -16157.414} C_VEL
LIN {X 0,Y 305.496,Z 250.432,A -85,B 0,C 180,E1 -16161.6,E2 -16161.6} C_VEL
LIN {X 0,Y 305.464,Z 250.433,A -85,B 0,C 180,E1 -16164.887,E2 -16164.887} C_VEL
LIN {X 0,Y 305.444,Z 250.434,A -85,B 0,C 180,E1 -16168.358,E2 -16168.358} C_VEL
LIN {X 0,Y 305.477,Z 250.433,A -85,B 0,C 180,E1 -16171.109,E2 -16171.109} C_VEL
LIN {X 0,Y 305.502,Z 250.428,A -85,B 0,C 180,E1 -16174.081,E2 -16174.081} C_VEL
LIN {X 0,Y 305.493,Z 250.432,A -85,B 0,C 180,E1 -16176.977,E2 -16176.977} C_VEL
LIN {X 0,Y 305.545,Z 250.426,A -85,B 0,C 180,E1 -16181.215,E2 -16181.215} C_VEL
LIN {X 0,Y 305.597,Z 250.418,A -85,B 0,C 180,E1 -16184.848,E2 -16184.848} C_VEL
LIN {X 0,Y 304.993,Z 250.499,A -85,B 0,C 180,E1 -16185.947,E2 -16185.947} C_VEL
LIN {X 0,Y 302.134,Z 250.856,A -85,B 0,C 180,E1 -16187.737,E2 -16187.737} C_VEL
LIN {X 0,Y 299.716,Z 251.153,A -85,B 0,C 180,E1 -16189.189,E2 -16189.189} C_VEL
LIN {X 0,Y 298.744,Z 251.272,A -85,B 0,C 180,E1 -16190.315,E2 -16190.315} C_VEL
LIN {X 0,Y 298.703,Z 251.276,A -85,B 0,C 180,E1 -16190.695,E2 -16190.695} C_VEL
LIN {X 0,Y 298.799,Z 251.264,A -85,B 0,C 180,E1 -16193.246,E2 -16193.246} C_VEL
LIN {X 0,Y 298.906,Z 251.254,A -85,B 0,C 180,E1 -16198.653,E2 -16198.653} C_VEL
LIN {X 0,Y 298.923,Z 251.248,A -85,B 0,C 180,E1 -16201.347,E2 -16201.347} C_VEL
LIN {X 0,Y 298.778,Z 251.267,A -85,B 0,C 180,E1 -16206.754,E2 -16206.754} C_VEL
LIN {X 0,Y 298.627,Z 251.284,A -85,B 0,C 180,E1 -16209.482,E2 -16209.482} C_VEL
LIN {X 0,Y 298.553,Z 251.294,A -85,B 0,C 180,E1 -16213.615,E2 -16213.615} C_VEL
LIN {X 0,Y 298.551,Z 251.296,A -85,B 0,C 180,E1 -16216.409,E2 -16216.409} C_VEL
LIN {X 0,Y 298.508,Z 251.302,A -85,B 0,C 180,E1 -16219.652,E2 -16219.652} C_VEL
LIN {X 0,Y 298.389,Z 251.319,A -85,B 0,C 180,E1 -16223.603,E2 -16223.603} C_VEL
LIN {X 0,Y 298.404,Z 251.316,A -85,B 0,C 180,E1 -16226.583,E2 -16226.583} C_VEL
LIN {X 0,Y 298.394,Z 251.321,A -85,B 0,C 180,E1 -16229.644,E2 -16229.644} C_VEL
LIN {X 0,Y 298.394,Z 251.318,A -85,B 0,C 180,E1 -16232.8,E2 -16232.8} C_VEL
LIN {X 0,Y 298.429,Z 251.312,A -85,B 0,C 180,E1 -16236.803,E2 -16236.803} C_VEL
LIN {X 0,Y 298.438,Z 251.446,A -85,B 0,C 180,E1 -16239.178,E2 -16239.178} C_VEL
LIN {X 0,Y 299.354,Z 256.29,A -85,B 0,C 180,E1 -16243.298,E2 -16243.298} C_VEL
LIN {X 0,Y 300.263,Z 261.315,A -85,B 0,C 180,E1 -16247.252,E2 -16247.252} C_VEL
LIN {X 0,Y 301.139,Z 266.375,A -85,B 0,C 180,E1 -16250.94,E2 -16250.94} C_VEL
LIN {X 0,Y 301.352,Z 270.15,A -85,B 0,C 180,E1 -16253.509,E2 -16253.509} C_VEL
LIN {X 0,Y 300.584,Z 275.108,A -85,B 0,C 180,E1 -16256.671,E2 -16256.671} C_VEL
LIN {X 0,Y 299.574,Z 281.233,A -85,B 0,C 180,E1 -16260.485,E2 -16260.485} C_VEL
LIN {X 0,Y 298.698,Z 287.267,A -85,B 0,C 180,E1 -16264.197,E2 -16264.197} C_VEL
LIN {X 0,Y 298.427,Z 289.279,A -85,B 0,C 180,E1 -16265.434,E2 -16265.434} C_VEL
LIN {X 0,Y 301.287,Z 302.704,A -85,B 0,C 180,E1 -16266.255,E2 -16266.255} C_VEL
LIN {X 0,Y 303.292,Z 316.282,A -85,B 0,C 180,E1 -16267.323,E2 -16267.323} C_VEL
LIN {X 0,Y 304.32,Z 328.385,A -85,B 0,C 180,E1 -16268.493,E2 -16268.493} C_VEL
LIN {X 0,Y 304.8,Z 337.759,A -85,B 0,C 180,E1 -16269.589,E2 -16269.589} C_VEL
LIN {X 0,Y 303.074,Z 349.034,A -85,B 0,C 180,E1 -16271.056,E2 -16271.056} C_VEL
LIN {X 0,Y 301.521,Z 358.769,A -85,B 0,C 180,E1 -16272.66,E2 -16272.66} C_VEL
LIN {X 0,Y 300.26,Z 367.256,A -85,B 0,C 180,E1 -16274.385,E2 -16274.385} C_VEL
LIN {X 0,Y 298.943,Z 375.324,A -85,B 0,C 180,E1 -16276.403,E2 -16276.403} C_VEL
LIN {X 0,Y 297.911,Z 381.801,A -85,B 0,C 180,E1 -16278.433,E2 -16278.433} C_VEL
LIN {X 0,Y 297.272,Z 386.959,A -85,B 0,C 180,E1 -16280.474,E2 -16280.474} C_VEL
LIN {X 0,Y 296.868,Z 390.971,A -85,B 0,C 180,E1 -16282.519,E2 -16282.519} C_VEL
LIN {X 0,Y 296.689,Z 393.942,A -85,B 0,C 180,E1 -16284.563,E2 -16284.563} C_VEL
LIN {X 0,Y 296.667,Z 395.36,A -85,B 0,C 180,E1 -16285.925,E2 -16285.925} C_VEL
LIN {X 0,Y 296.669,Z 396.991,A -85,B 0,C 180,E1 -16288.643,E2 -16288.643} C_VEL
LIN {X 0,Y 296.781,Z 397.215,A -85,B 0,C 180,E1 -16290,E2 -16290} C_VEL
LIN {X 0,Y 296.669,Z 396.986,A -85,B 0,C 180,E1 -16291.358,E2 -16291.358} C_VEL
LIN {X 0,Y 296.666,Z 395.352,A -85,B 0,C 180,E1 -16294.076,E2 -16294.076} C_VEL
LIN {X 0,Y 296.738,Z 393.345,A -85,B 0,C 180,E1 -16295.88,E2 -16295.88} C_VEL
LIN {X 0,Y 296.963,Z 389.705,A -85,B 0,C 180,E1 -16298.164,E2 -16298.164} C_VEL
LIN {X 0,Y 297.459,Z 385.315,A -85,B 0,C 180,E1 -16300.207,E2 -16300.207} C_VEL
LIN {X 0,Y 298.185,Z 379.731,A -85,B 0,C 180,E1 -16302.247,E2 -16302.247} C_VEL
LIN {X 0,Y 299.385,Z 372.784,A -85,B 0,C 180,E1 -16304.27,E2 -16304.27} C_VEL
LIN {X 0,Y 300.562,Z 365.694,A -85,B 0,C 180,E1 -16305.947,E2 -16305.947} C_VEL
LIN {X 0,Y 301.782,Z 357.145,A -85,B 0,C 180,E1 -16307.623,E2 -16307.623} C_VEL
LIN {X 0,Y 303.266,Z 347.79,A -85,B 0,C 180,E1 -16309.108,E2 -16309.108} C_VEL
LIN {X 0,Y 304.781,Z 337.628,A -85,B 0,C 180,E1 -16310.412,E2 -16310.412} C_VEL
LIN {X 0,Y 304.1,Z 325.579,A -85,B 0,C 180,E1 -16311.785,E2 -16311.785} C_VEL
LIN {X 0,Y 303.037,Z 314.184,A -85,B 0,C 180,E1 -16312.844,E2 -16312.844} C_VEL
LIN {X 0,Y 300.901,Z 300.869,A -85,B 0,C 180,E1 -16313.851,E2 -16313.851} C_VEL
LIN {X 0,Y 298.444,Z 289.219,A -85,B 0,C 180,E1 -16314.552,E2 -16314.552} C_VEL
LIN {X 0,Y 299.388,Z 282.42,A -85,B 0,C 180,E1 -16318.766,E2 -16318.766} C_VEL
LIN {X 0,Y 300.355,Z 276.227,A -85,B 0,C 180,E1 -16322.609,E2 -16322.609} C_VEL
LIN {X 0,Y 301.216,Z 271.367,A -85,B 0,C 180,E1 -16325.684,E2 -16325.684} C_VEL
LIN {X 0,Y 301.298,Z 267.497,A -85,B 0,C 180,E1 -16328.227,E2 -16328.227} C_VEL
LIN {X 0,Y 300.539,Z 262.793,A -85,B 0,C 180,E1 -16331.556,E2 -16331.556} C_VEL
LIN {X 0,Y 299.634,Z 257.948,A -85,B 0,C 180,E1 -16335.279,E2 -16335.279} C_VEL
LIN {X 0,Y 298.812,Z 253.685,A -85,B 0,C 180,E1 -16338.82,E2 -16338.82} C_VEL
LIN {X 0,Y 298.417,Z 251.313,A -85,B 0,C 180,E1 -16341.004,E2 -16341.004} C_VEL
LIN {X 0,Y 298.408,Z 251.316,A -85,B 0,C 180,E1 -16343.929,E2 -16343.929} C_VEL
LIN {X 0,Y 298.396,Z 251.315,A -85,B 0,C 180,E1 -16347.2,E2 -16347.2} C_VEL
LIN {X 0,Y 298.405,Z 251.315,A -85,B 0,C 180,E1 -16350.625,E2 -16350.625} C_VEL
LIN {X 0,Y 298.425,Z 251.312,A -85,B 0,C 180,E1 -16354.919,E2 -16354.919} C_VEL
LIN {X 0,Y 298.436,Z 251.31,A -85,B 0,C 180,E1 -16359.314,E2 -16359.314} C_VEL
LIN {X 0,Y 298.538,Z 251.3,A -85,B 0,C 180,E1 -16362.179,E2 -16362.179} C_VEL
LIN {X 0,Y 298.597,Z 251.289,A -85,B 0,C 180,E1 -16364.995,E2 -16364.995} C_VEL
LIN {X 0,Y 298.586,Z 251.29,A -85,B 0,C 180,E1 -16369.146,E2 -16369.146} C_VEL
LIN {X 0,Y 298.78,Z 251.267,A -85,B 0,C 180,E1 -16373.246,E2 -16373.246} C_VEL
LIN {X 0,Y 298.925,Z 251.248,A -85,B 0,C 180,E1 -16378.653,E2 -16378.653} C_VEL
LIN {X 0,Y 298.908,Z 251.253,A -85,B 0,C 180,E1 -16381.347,E2 -16381.347} C_VEL
LIN {X 0,Y 298.771,Z 251.267,A -85,B 0,C 180,E1 -16386.755,E2 -16386.755} C_VEL
LIN {X 0,Y 298.629,Z 251.287,A -85,B 0,C 180,E1 -16389.482,E2 -16389.482} C_VEL
LIN {X 0,Y 298.55,Z 251.295,A -85,B 0,C 180,E1 -16393.616,E2 -16393.616} C_VEL
LIN {X 0,Y 298.49,Z 251.303,A -85,B 0,C 180,E1 -16396.412,E2 -16396.412} C_VEL
LIN {X 0,Y 298.486,Z 251.302,A -85,B 0,C 180,E1 -16399.639,E2 -16399.639} C_VEL
LIN {X 0,Y 298.424,Z 251.309,A -85,B 0,C 180,E1 -16403.601,E2 -16403.601} C_VEL
LIN {X 0,Y 298.411,Z 251.315,A -85,B 0,C 180,E1 -16406.582,E2 -16406.582} C_VEL
LIN {X 0,Y 298.397,Z 251.313,A -85,B 0,C 180,E1 -16409.644,E2 -16409.644} C_VEL
LIN {X 0,Y 298.396,Z 251.315,A -85,B 0,C 180,E1 -16412.8,E2 -16412.8} C_VEL
LIN {X 0,Y 298.45,Z 251.308,A -85,B 0,C 180,E1 -16416.807,E2 -16416.807} C_VEL
LIN {X 0,Y 298.412,Z 251.31,A -85,B 0,C 180,E1 -16419.486,E2 -16419.486} C_VEL
LIN {X 0,Y 298.401,Z 251.313,A -85,B 0,C 180,E1 -16423.103,E2 -16423.103} C_VEL
LIN {X 0,Y 298.406,Z 251.312,A -85,B 0,C 180,E1 -16426.921,E2 -16426.921} C_VEL
LIN {X 0,Y 298.391,Z 251.314,A -85,B 0,C 180,E1 -16431.01,E2 -16431.01} C_VEL
LIN {X 0,Y 298.303,Z 251.328,A -85,B 0,C 180,E1 -16433.913,E2 -16433.913} C_VEL
LIN {X 0,Y 298.159,Z 251.345,A -85,B 0,C 180,E1 -16435.589,E2 -16435.589} C_VEL
LIN {X 0,Y 297.989,Z 251.649,A -85,B 0,C 180,E1 -16437.149,E2 -16437.149} C_VEL
LIN {X 0,Y 297.883,Z 254.458,A -85,B 0,C 180,E1 -16440.803,E2 -16440.803} C_VEL
LIN {X 0,Y 297.742,Z 257.86,A -85,B 0,C 180,E1 -16444.857,E2 -16444.857} C_VEL
LIN {X 0,Y 297.749,Z 258.417,A -85,B 0,C 180,E1 -16445.501,E2 -16445.501} C_VEL
LIN {X 0,Y 302.102,Z 271.536,A -85,B 0,C 180,E1 -16446.517,E2 -16446.517} C_VEL
LIN {X 0,Y 305.382,Z 283.639,A -85,B 0,C 180,E1 -16447.649,E2 -16447.649} C_VEL
LIN {X 0,Y 307.375,Z 293.434,A -85,B 0,C 180,E1 -16448.717,E2 -16448.717} C_VEL
LIN {X 0,Y 306.291,Z 304.138,A -85,B 0,C 180,E1 -16449.868,E2 -16449.868} C_VEL
LIN {X 0,Y 305.03,Z 313.979,A -85,B 0,C 180,E1 -16451.182,E2 -16451.182} C_VEL
